METHOD FB_init : BOOL
VAR_INPUT
	bInitRetains : BOOL; // if TRUE, the retain variables are initialized (warm start / cold start)
	bInCopyCode : BOOL;  // if TRUE, the instance afterwards gets moved into the copy code (online change)
	InitialValue : ETcVnMorphologicalOperator;
END_VAR
localData := InitialValue;
AddBaseDatatype(enumBaseDatatype);
ClearReference();

AddLocalEnumeration('TCVN_MO_EROSION', ETcVnMorphologicalOperator.TCVN_MO_EROSION);
AddLocalEnumeration('TCVN_MO_DILATION', ETcVnMorphologicalOperator.TCVN_MO_DILATION);
AddLocalEnumeration('TCVN_MO_OPENING', ETcVnMorphologicalOperator.TCVN_MO_OPENING);
AddLocalEnumeration('TCVN_MO_CLOSING', ETcVnMorphologicalOperator.TCVN_MO_CLOSING);
AddLocalEnumeration('TCVN_MO_GRADIENT', ETcVnMorphologicalOperator.TCVN_MO_GRADIENT);
AddLocalEnumeration('TCVN_MO_WHITE_TOPHAT', .TCVN_MO_WHITE_TOPHAT);
AddLocalEnumeration('TCVN_MO_BLACK_TOPHAT', ETcVnMorphologicalOperator.TCVN_MO_BLACK_TOPHAT);
AddLocalEnumeration('TCVN_MO_OPENING_BY_RECONSTRUCTION', ETcVnMorphologicalOperator.TCVN_MO_OPENING_BY_RECONSTRUCTION);
AddLocalEnumeration('TCVN_MO_CLOSING_BY_RECONSTRUCTION', ETcVnMorphologicalOperator.TCVN_MO_CLOSING_BY_RECONSTRUCTION);
AddLocalEnumeration('TCVN_MO_WHITE_TOPHAT_BY_RECONSTRUCTION', ETcVnMorphologicalOperator.TCVN_MO_WHITE_TOPHAT_BY_RECONSTRUCTION);
AddLocalEnumeration('TCVN_MO_BLACK_TOPHAT_BY_RECONSTRUCTION', ETcVnMorphologicalOperator.TCVN_MO_BLACK_TOPHAT_BY_RECONSTRUCTION);
END_METHOD

PROPERTY PUBLIC Identifier : T_MAXSTRING
GET
Identifier := 'ETcVnMorphologicalOperator';
END_GET
END_PROPERTY

METHOD IsEnumeratorValueEqual : BOOL
VAR_INPUT
	Enumerator : I_KeyValueForwardEnumerator;
END_VAR
VAR
	storedValue : ETcVnMorphologicalOperator;
END_VAR
IF NOT Enumerator.TryGet(storedValue) THEN
	RETURN;
END_IF

IsEnumeratorValueEqual := storedValue = activeData;
END_METHOD

METHOD PUBLIC MakeReferenceTo
VAR_INPUT
	ReferenceTarget : REFERENCE TO ETcVnMorphologicalOperator;
END_VAR
activeData REF= ReferenceTarget;
SetBaseDatatypeReference();
END_METHOD

METHOD PROTECTED SetBaseDatatypeReference
VAR_INPUT
END_VAR
enumBaseDatatype.MakeReferenceTo(activeData);
END_METHOD

PROPERTY PUBLIC Size : UDINT
GET
Size := SIZEOF(activeData);
END_GET
END_PROPERTY

METHOD TryMakeReferenceTo : BOOL
VAR_INPUT
	Target : I_Datatype;
END_VAR
VAR
	targetAsEnum : I_EnumDatatype;
	pTargetData : POINTER TO ETcVnMorphologicalOperator;
END_VAR
IF NOT Target.TryResolveAsEnumDatatype(targetAsEnum) THEN
	RETURN;
END_IF

IF targetAsEnum.Identifier <> Identifier THEN
	RETURN;
END_IF

pTargetData := Target.Address;
activeData REF= pTargetData^;
SetBaseDatatypeReference();
TryMakeReferenceTo := TRUE;
END_METHOD

PROPERTY PUBLIC Value : ETcVnMorphologicalOperator
GET
Value := activeData;
END_GET
SET
activeData := Value;
END_SET
END_PROPERTY

END_FUNCTION_BLOCK

// ---- Enums/_ETcVnNbc.TcPOU
{attribute 'linkalways'} 
{attribute 'no_explicit_call' := 'This FB is a CLASS and must be accessed using methods or properties'}
{attribute 'enable_dynamic_creation'}
FUNCTION_BLOCK _ETcVnNbc EXTENDS EnumDatatypeBase
VAR
	localData : ETcVnNbc;
	activeData : REFERENCE TO ETcVnNbc;
	enumBaseDatatype : _UDINT(localData);
END_VAR

METHOD PRIVATE AddLocalEnumeration
VAR_INPUT
	Enumeration : T_MAXSTRING;
	Value : ETcVnNbc;
END_VAR
AddEnumeration(Enumeration, Value);
END_METHOD

PROPERTY PUBLIC Address : PVOID
GET
Address := ADR(activeData);
END_GET
END_PROPERTY

METHOD PUBLIC ClearReference
VAR_INPUT
END_VAR
activeData REF= localData;
SetBaseDatatypeReference();
END_METHOD

METHOD PUBLIC Clone : I_Datatype
VAR
    pClone : POINTER TO _ETcVnNbc;
END_VAR
pClone := __NEW(_ETcVnNbc(InitialValue := Value));
Clone := pClone^;
END_METHOD

METHOD FB_init : BOOL
VAR_INPUT
	bInitRetains : BOOL; // if TRUE, the retain variables are initialized (warm start / cold start)
	bInCopyCode : BOOL;  // if TRUE, the instance afterwards gets moved into the copy code (online change)
	InitialValue : ETcVnNbc;
END_VAR
localData := InitialValue;
AddBaseDatatype(enumBaseDatatype);
ClearReference();

AddLocalEnumeration('TCVN_NBC_CLASSIFIER', ETcVnNbc.TCVN_NBC_CLASSIFIER);
AddLocalEnumeration('TCVN_NBC_NOVELTY_DETECTOR', ETcVnNbc.TCVN_NBC_NOVELTY_DETECTOR);
END_METHOD

PROPERTY PUBLIC Identifier : T_MAXSTRING
GET
Identifier := 'ETcVnNbc';
END_GET
END_PROPERTY

METHOD IsEnumeratorValueEqual : BOOL
VAR_INPUT
	Enumerator : I_KeyValueForwardEnumerator;
END_VAR
VAR
	storedValue : ETcVnNbc;
END_VAR
IF NOT Enumerator.TryGet(storedValue) THEN
	RETURN;
END_IF

IsEnumeratorValueEqual := storedValue = activeData;
END_METHOD

METHOD PUBLIC MakeReferenceTo
VAR_INPUT
	ReferenceTarget : REFERENCE TO ETcVnNbc;
END_VAR
activeData REF= ReferenceTarget;
SetBaseDatatypeReference();
END_METHOD

METHOD PROTECTED SetBaseDatatypeReference
VAR_INPUT
END_VAR
enumBaseDatatype.MakeReferenceTo(activeData);
END_METHOD

PROPERTY PUBLIC Size : UDINT
GET
Size := SIZEOF(activeData);
END_GET
END_PROPERTY

METHOD TryMakeReferenceTo : BOOL
VAR_INPUT
	Target : I_Datatype;
END_VAR
VAR
	targetAsEnum : I_EnumDatatype;
	pTargetData : POINTER TO ETcVnNbc;
END_VAR
IF NOT Target.TryResolveAsEnumDatatype(targetAsEnum) THEN
	RETURN;
END_IF

IF targetAsEnum.Identifier <> Identifier THEN
	RETURN;
END_IF

pTargetData := Target.Address;
activeData REF= pTargetData^;
SetBaseDatatypeReference();
TryMakeReferenceTo := TRUE;
END_METHOD

PROPERTY PUBLIC Value : ETcVnNbc
GET
Value := activeData;
END_GET
SET
activeData := Value;
END_SET
END_PROPERTY

END_FUNCTION_BLOCK

// ---- Enums/_ETcVnNormalizationType.TcPOU
{attribute 'linkalways'} 
{attribute 'no_explicit_call' := 'This FB is a CLASS and must be accessed using methods or properties'}
{attribute 'enable_dynamic_creation'}
FUNCTION_BLOCK _ETcVnNormalizationType EXTENDS EnumDatatypeBase
VAR
	localData : ETcVnNormalizationType;
	activeData : REFERENCE TO ETcVnNormalizationType;
	enumBaseDatatype : _DINT(localData);
END_VAR

METHOD PRIVATE AddLocalEnumeration
VAR_INPUT
	Enumeration : T_MAXSTRING;
	Value : ETcVnNormalizationType;
END_VAR
AddEnumeration(Enumeration, Value);
END_METHOD

PROPERTY PUBLIC Address : PVOID
GET
Address := ADR(activeData);
END_GET
END_PROPERTY

METHOD PUBLIC ClearReference
VAR_INPUT
END_VAR
activeData REF= localData;
SetBaseDatatypeReference();
END_METHOD

METHOD PUBLIC Clone : I_Datatype
VAR
    pClone : POINTER TO _ETcVnNormalizationType;
END_VAR
pClone := __NEW(_ETcVnNormalizationType(InitialValue := Value));
Clone := pClone^;
END_METHOD

METHOD FB_init : BOOL
VAR_INPUT
	bInitRetains : BOOL; // if TRUE, the retain variables are initialized (warm start / cold start)
	bInCopyCode : BOOL;  // if TRUE, the instance afterwards gets moved into the copy code (online change)
	InitialValue : ETcVnNormalizationType;
END_VAR
localData := InitialValue;
AddBaseDatatype(enumBaseDatatype);
ClearReference();

AddLocalEnumeration('TCVN_NT_INF', ETcVnNormalizationType.TCVN_NT_INF);
AddLocalEnumeration('TCVN_NT_L1', ETcVnNormalizationType.TCVN_NT_L1);
AddLocalEnumeration('TCVN_NT_L2', ETcVnNormalizationType.TCVN_NT_L2);
AddLocalEnumeration('TCVN_NT_L2SQR', ETcVnNormalizationType.TCVN_NT_L2SQR);
AddLocalEnumeration('TCVN_NT_HAMMING', ETcVnNormalizationType.TCVN_NT_HAMMING);
AddLocalEnumeration('TCVN_NT_HAMMING2', ETcVnNormalizationType.TCVN_NT_HAMMING2);
AddLocalEnumeration('TCVN_NT_RELATIVE_INF', ETcVnNormalizationType.TCVN_NT_RELATIVE_INF);
AddLocalEnumeration('TCVN_NT_RELATIVE_L1', ETcVnNormalizationType.TCVN_NT_RELATIVE_L1);
AddLocalEnumeration('TCVN_NT_RELATIVE_L2', ETcVnNormalizationType.TCVN_NT_RELATIVE_L2);
AddLocalEnumeration('TCVN_NT_RELATIVE_L2SQR', ETcVnNormalizationType.TCVN_NT_RELATIVE_L2SQR);
AddLocalEnumeration('TCVN_NT_RELATIVE_HAMMING', ETcVnNormalizationType.TCVN_NT_RELATIVE_HAMMING);
AddLocalEnumeration('TCVN_NT_RELATIVE_HAMMING2', ETcVnNormalizationType.TCVN_NT_RELATIVE_HAMMING2);
AddLocalEnumeration('TCVN_NT_MINMAX', ETcVnNormalizationType.TCVN_NT_MINMAX);
END_METHOD

PROPERTY PUBLIC Identifier : T_MAXSTRING
GET
Identifier := 'ETcVnNormalizationType';
END_GET
END_PROPERTY

METHOD IsEnumeratorValueEqual : BOOL
VAR_INPUT
	Enumerator : I_KeyValueForwardEnumerator;
END_VAR
VAR
	storedValue : ETcVnNormalizationType;
END_VAR
IF NOT Enumerator.TryGet(storedValue) THEN
	RETURN;
END_IF

IsEnumeratorValueEqual := storedValue = activeData;
END_METHOD

METHOD PUBLIC MakeReferenceTo
VAR_INPUT
	ReferenceTarget : REFERENCE TO ETcVnNormalizationType;
END_VAR
activeData REF= ReferenceTarget;
SetBaseDatatypeReference();
END_METHOD

METHOD PROTECTED SetBaseDatatypeReference
VAR_INPUT
END_VAR
enumBaseDatatype.MakeReferenceTo(activeData);
END_METHOD

PROPERTY PUBLIC Size : UDINT
GET
Size := SIZEOF(activeData);
END_GET
END_PROPERTY

METHOD TryMakeReferenceTo : BOOL
VAR_INPUT
	Target : I_Datatype;
END_VAR
VAR
	targetAsEnum : I_EnumDatatype;
	pTargetData : POINTER TO ETcVnNormalizationType;
END_VAR
IF NOT Target.TryResolveAsEnumDatatype(targetAsEnum) THEN
	RETURN;
END_IF

IF targetAsEnum.Identifier <> Identifier THEN
	RETURN;
END_IF

pTargetData := Target.Address;
activeData REF= pTargetData^;
SetBaseDatatypeReference();
TryMakeReferenceTo := TRUE;
END_METHOD

PROPERTY PUBLIC Value : ETcVnNormalizationType
GET
Value := activeData;
END_GET
SET
activeData := Value;
END_SET
END_PROPERTY

END_FUNCTION_BLOCK

// ---- Enums/_ETcVnOcrModelType.TcPOU
{attribute 'linkalways'} 
{attribute 'no_explicit_call' := 'This FB is a CLASS and must be accessed using methods or properties'}
{attribute 'enable_dynamic_creation'}
FUNCTION_BLOCK _ETcVnOcrModelType EXTENDS EnumDatatypeBase
VAR
	localData : ETcVnOcrModelType;
	activeData : REFERENCE TO ETcVnOcrModelType;
	enumBaseDatatype : _ULINT(localData);
END_VAR

METHOD PRIVATE AddLocalEnumeration
VAR_INPUT
	Enumeration : T_MAXSTRING;
	Value : ETcVnOcrModelType;
END_VAR
AddEnumeration(Enumeration, Value);
END_METHOD

PROPERTY PUBLIC Address : PVOID
GET
Address := ADR(activeData);
END_GET
END_PROPERTY

METHOD PUBLIC ClearReference
VAR_INPUT
END_VAR
activeData REF= localData;
SetBaseDatatypeReference();
END_METHOD

METHOD PUBLIC Clone : I_Datatype
VAR
    pClone : POINTER TO _ETcVnOcrModelType;
END_VAR
pClone := __NEW(_ETcVnOcrModelType(InitialValue := Value));
Clone := pClone^;
END_METHOD

METHOD FB_init : BOOL
VAR_INPUT
	bInitRetains : BOOL; // if TRUE, the retain variables are initialized (warm start / cold start)
	bInCopyCode : BOOL;  // if TRUE, the instance afterwards gets moved into the copy code (online change)
	InitialValue : ETcVnOcrModelType;
END_VAR
localData := InitialValue;
AddBaseDatatype(enumBaseDatatype);
ClearReference();

AddLocalEnumeration('TCVN_OMT_NUMBERS', ETcVnOcrModelType.TCVN_OMT_NUMBERS);
AddLocalEnumeration('TCVN_OMT_NUMBERS_SC', ETcVnOcrModelType.TCVN_OMT_NUMBERS_SC);
AddLocalEnumeration('TCVN_OMT_UCLETTERS', ETcVnOcrModelType.TCVN_OMT_UCLETTERS);
AddLocalEnumeration('TCVN_OMT_NUMBERS_SC_UCLETTERS', ETcVnOcrModelType.TCVN_OMT_NUMBERS_SC_UCLETTERS);
END_METHOD

PROPERTY PUBLIC Identifier : T_MAXSTRING
GET
Identifier := 'ETcVnOcrModelType';
END_GET
END_PROPERTY

METHOD IsEnumeratorValueEqual : BOOL
VAR_INPUT
	Enumerator : I_KeyValueForwardEnumerator;
END_VAR
VAR
	storedValue : ETcVnOcrModelType;
END_VAR
IF NOT Enumerator.TryGet(storedValue) THEN
	RETURN;
END_IF

IsEnumeratorValueEqual := storedValue = activeData;
END_METHOD

METHOD PUBLIC MakeReferenceTo
VAR_INPUT
	ReferenceTarget : REFERENCE TO ETcVnOcrModelType;
END_VAR
activeData REF= ReferenceTarget;
SetBaseDatatypeReference();
END_METHOD

METHOD PROTECTED SetBaseDatatypeReference
VAR_INPUT
END_VAR
enumBaseDatatype.MakeReferenceTo(activeData);
END_METHOD

PROPERTY PUBLIC Size : UDINT
GET
Size := SIZEOF(activeData);
END_GET
END_PROPERTY

METHOD TryMakeReferenceTo : BOOL
VAR_INPUT
	Target : I_Datatype;
END_VAR
VAR
	targetAsEnum : I_EnumDatatype;
	pTargetData : POINTER TO ETcVnOcrModelType;
END_VAR
IF NOT Target.TryResolveAsEnumDatatype(targetAsEnum) THEN
	RETURN;
END_IF

IF targetAsEnum.Identifier <> Identifier THEN
	RETURN;
END_IF

pTargetData := Target.Address;
activeData REF= pTargetData^;
SetBaseDatatypeReference();
TryMakeReferenceTo := TRUE;
END_METHOD

PROPERTY PUBLIC Value : ETcVnOcrModelType
GET
Value := activeData;
END_GET
SET
activeData := Value;
END_SET
END_PROPERTY

END_FUNCTION_BLOCK

// ---- Enums/_ETcVnOcrOptions.TcPOU
{attribute 'linkalways'} 
{attribute 'no_explicit_call' := 'This FB is a CLASS and must be accessed using methods or properties'}
{attribute 'enable_dynamic_creation'}
FUNCTION_BLOCK _ETcVnOcrOptions EXTENDS EnumDatatypeBase
VAR
	localData : ETcVnOcrOptions;
	activeData : REFERENCE TO ETcVnOcrOptions;
	enumBaseDatatype : _UDINT(localData);
END_VAR

METHOD PRIVATE AddLocalEnumeration
VAR_INPUT
	Enumeration : T_MAXSTRING;
	Value : ETcVnOcrOptions;
END_VAR
AddEnumeration(Enumeration, Value);
END_METHOD

PROPERTY PUBLIC Address : PVOID
GET
Address := ADR(activeData);
END_GET
END_PROPERTY

METHOD PUBLIC ClearReference
VAR_INPUT
END_VAR
activeData REF= localData;
SetBaseDatatypeReference();
END_METHOD

METHOD PUBLIC Clone : I_Datatype
VAR
    pClone : POINTER TO _ETcVnOcrOptions;
END_VAR
pClone := __NEW(_ETcVnOcrOptions(InitialValue := Value));
Clone := pClone^;
END_METHOD

METHOD FB_init : BOOL
VAR_INPUT
	bInitRetains : BOOL; // if TRUE, the retain variables are initialized (warm start / cold start)
	bInCopyCode : BOOL;  // if TRUE, the instance afterwards gets moved into the copy code (online change)
	InitialValue : ETcVnOcrOptions;
END_VAR
localData := InitialValue;
AddBaseDatatype(enumBaseDatatype);
ClearReference();

AddLocalEnumeration('TCVN_OO_WITHBLANKS', ETcVnOcrOptions.TCVN_OO_WITHBLANKS);
END_METHOD

PROPERTY PUBLIC Identifier : T_MAXSTRING
GET
Identifier := 'ETcVnOcrOptions';
END_GET
END_PROPERTY

METHOD IsEnumeratorValueEqual : BOOL
VAR_INPUT
	Enumerator : I_KeyValueForwardEnumerator;
END_VAR
VAR
	storedValue : ETcVnOcrOptions;
END_VAR
IF NOT Enumerator.TryGet(storedValue) THEN
	RETURN;
END_IF

IsEnumeratorValueEqual := storedValue = activeData;
END_METHOD

METHOD PUBLIC MakeReferenceTo
VAR_INPUT
	ReferenceTarget : REFERENCE TO ETcVnOcrOptions;
END_VAR
activeData REF= ReferenceTarget;
SetBaseDatatypeReference();
END_METHOD

METHOD PROTECTED SetBaseDatatypeReference
VAR_INPUT
END_VAR
enumBaseDatatype.MakeReferenceTo(activeData);
END_METHOD

PROPERTY PUBLIC Size : UDINT
GET
Size := SIZEOF(activeData);
END_GET
END_PROPERTY

METHOD TryMakeReferenceTo : BOOL
VAR_INPUT
	Target : I_Datatype;
END_VAR
VAR
	targetAsEnum : I_EnumDatatype;
	pTargetData : POINTER TO ETcVnOcrOptions;
END_VAR
IF NOT Target.TryResolveAsEnumDatatype(targetAsEnum) THEN
	RETURN;
END_IF

IF targetAsEnum.Identifier <> Identifier THEN
	RETURN;
END_IF

pTargetData := Target.Address;
activeData REF= pTargetData^;
SetBaseDatatypeReference();
TryMakeReferenceTo := TRUE;
END_METHOD

PROPERTY PUBLIC Value : ETcVnOcrOptions
GET
Value := activeData;
END_GET
SET
activeData := Value;
END_SET
END_PROPERTY

END_FUNCTION_BLOCK

// ---- Enums/_ETcVnOrientationMethod.TcPOU
{attribute 'linkalways'} 
{attribute 'no_explicit_call' := 'This FB is a CLASS and must be accessed using methods or properties'}
{attribute 'enable_dynamic_creation'}
FUNCTION_BLOCK _ETcVnOrientationMethod EXTENDS EnumDatatypeBase
VAR
	localData : ETcVnOrientationMethod;
	activeData : REFERENCE TO ETcVnOrientationMethod;
	enumBaseDatatype : _DINT(localData);
END_VAR

METHOD PRIVATE AddLocalEnumeration
VAR_INPUT
	Enumeration : T_MAXSTRING;
	Value : ETcVnOrientationMethod;
END_VAR
AddEnumeration(Enumeration, Value);
END_METHOD

PROPERTY PUBLIC Address : PVOID
GET
Address := ADR(activeData);
END_GET
END_PROPERTY

METHOD PUBLIC ClearReference
VAR_INPUT
END_VAR
activeData REF= localData;
SetBaseDatatypeReference();
END_METHOD

METHOD PUBLIC Clone : I_Datatype
VAR
    pClone : POINTER TO _ETcVnOrientationMethod;
END_VAR
pClone := __NEW(_ETcVnOrientationMethod(InitialValue := Value));
Clone := pClone^;
END_METHOD

METHOD FB_init : BOOL
VAR_INPUT
	bInitRetains : BOOL; // if TRUE, the retain variables are initialized (warm start / cold start)
	bInCopyCode : BOOL;  // if TRUE, the instance afterwards gets moved into the copy code (online change)
	InitialValue : ETcVnOrientationMethod;
END_VAR
localData := InitialValue;
AddBaseDatatype(enumBaseDatatype);
ClearReference();

AddLocalEnumeration('TCVN_OM_PCA', ETcVnOrientationMethod.TCVN_OM_PCA);
AddLocalEnumeration('TCVN_OM_FITELLIPSE', ETcVnOrientationMethod.TCVN_OM_FITELLIPSE);
AddLocalEnumeration('TCVN_OM_MOMENTS', ETcVnOrientationMethod.TCVN_OM_MOMENTS);
AddLocalEnumeration('TCVN_OM_ENCLOSINGRECT', ETcVnOrientationMethod.TCVN_OM_ENCLOSINGRECT);
END_METHOD

PROPERTY PUBLIC Identifier : T_MAXSTRING
GET
Identifier := 'ETcVnOrientationMethod';
END_GET
END_PROPERTY

METHOD IsEnumeratorValueEqual : BOOL
VAR_INPUT
	Enumerator : I_KeyValueForwardEnumerator;
END_VAR
VAR
	storedValue : ETcVnOrientationMethod;
END_VAR
IF NOT Enumerator.TryGet(storedValue) THEN
	RETURN;
END_IF

IsEnumeratorValueEqual := storedValue = activeData;
END_METHOD

METHOD PUBLIC MakeReferenceTo
VAR_INPUT
	ReferenceTarget : REFERENCE TO ETcVnOrientationMethod;
END_VAR
activeData REF= ReferenceTarget;
SetBaseDatatypeReference();
END_METHOD

METHOD PROTECTED SetBaseDatatypeReference
VAR_INPUT
END_VAR
enumBaseDatatype.MakeReferenceTo(activeData);
END_METHOD

PROPERTY PUBLIC Size : UDINT
GET
Size := SIZEOF(activeData);
END_GET
END_PROPERTY

METHOD TryMakeReferenceTo : BOOL
VAR_INPUT
	Target : I_Datatype;
END_VAR
VAR
	targetAsEnum : I_EnumDatatype;
	pTargetData : POINTER TO ETcVnOrientationMethod;
END_VAR
IF NOT Target.TryResolveAsEnumDatatype(targetAsEnum) THEN
	RETURN;
END_IF

IF targetAsEnum.Identifier <> Identifier THEN
	RETURN;
END_IF

pTargetData := Target.Address;
activeData REF= pTargetData^;
SetBaseDatatypeReference();
TryMakeReferenceTo := TRUE;
END_METHOD

PROPERTY PUBLIC Value : ETcVnOrientationMethod
GET
Value := activeData;
END_GET
SET
activeData := Value;
END_SET
END_PROPERTY

END_FUNCTION_BLOCK

// ---- Enums/_ETcVnPaddingMode.TcPOU
{attribute 'linkalways'} 
{attribute 'no_explicit_call' := 'This FB is a CLASS and must be accessed using methods or properties'}
{attribute 'enable_dynamic_creation'}
FUNCTION_BLOCK _ETcVnPaddingMode EXTENDS EnumDatatypeBase
VAR
	localData : ETcVnPaddingMode;
	activeData : REFERENCE TO ETcVnPaddingMode;
	enumBaseDatatype : _DINT(localData);
END_VAR

METHOD PRIVATE AddLocalEnumeration
VAR_INPUT
	Enumeration : T_MAXSTRING;
	Value : ETcVnPaddingMode;
END_VAR
AddEnumeration(Enumeration, Value);
END_METHOD

PROPERTY PUBLIC Address : PVOID
GET
Address := ADR(activeData);
END_GET
END_PROPERTY

METHOD PUBLIC ClearReference
VAR_INPUT
END_VAR
activeData REF= localData;
SetBaseDatatypeReference();
END_METHOD

METHOD PUBLIC Clone : I_Datatype
VAR
    pClone : POINTER TO _ETcVnPaddingMode;
END_VAR
pClone := __NEW(_ETcVnPaddingMode(InitialValue := Value));
Clone := pClone^;
END_METHOD

METHOD FB_init : BOOL
VAR_INPUT
	bInitRetains : BOOL; // if TRUE, the retain variables are initialized (warm start / cold start)
	bInCopyCode : BOOL;  // if TRUE, the instance afterwards gets moved into the copy code (online change)
	InitialValue : ETcVnPaddingMode;
END_VAR
localData := InitialValue;
AddBaseDatatype(enumBaseDatatype);
ClearReference();

AddLocalEnumeration('TCVN_PM_NONE', ETcVnPaddingMode.TCVN_PM_NONE);
AddLocalEnumeration('TCVN_PM_CROP_CENTER', ETcVnPaddingMode.TCVN_PM_CROP_CENTER);
AddLocalEnumeration('TCVN_PM_LETTERBOX', ETcVnPaddingMode.TCVN_PM_LETTERBOX);
END_METHOD

PROPERTY PUBLIC Identifier : T_MAXSTRING
GET
Identifier := 'ETcVnPaddingMode';
END_GET
END_PROPERTY

METHOD IsEnumeratorValueEqual : BOOL
VAR_INPUT
	Enumerator : I_KeyValueForwardEnumerator;
END_VAR
VAR
	storedValue : ETcVnPaddingMode;
END_VAR
IF NOT Enumerator.TryGet(storedValue) THEN
	RETURN;
END_IF

IsEnumeratorValueEqual := storedValue = activeData;
END_METHOD

METHOD PUBLIC MakeReferenceTo
VAR_INPUT
	ReferenceTarget : REFERENCE TO ETcVnPaddingMode;
END_VAR
activeData REF= ReferenceTarget;
SetBaseDatatypeReference();
END_METHOD

METHOD PROTECTED SetBaseDatatypeReference
VAR_INPUT
END_VAR
enumBaseDatatype.MakeReferenceTo(activeData);
END_METHOD

PROPERTY PUBLIC Size : UDINT
GET
Size := SIZEOF(activeData);
END_GET
END_PROPERTY

METHOD TryMakeReferenceTo : BOOL
VAR_INPUT
	Target : I_Datatype;
END_VAR
VAR
	targetAsEnum : I_EnumDatatype;
	pTargetData : POINTER TO ETcVnPaddingMode;
END_VAR
IF NOT Target.TryResolveAsEnumDatatype(targetAsEnum) THEN
	RETURN;
END_IF

IF targetAsEnum.Identifier <> Identifier THEN
	RETURN;
END_IF

pTargetData := Target.Address;
activeData REF= pTargetData^;
SetBaseDatatypeReference();
TryMakeReferenceTo := TRUE;
END_METHOD

PROPERTY PUBLIC Value : ETcVnPaddingMode
GET
Value := activeData;
END_GET
SET
activeData := Value;
END_SET
END_PROPERTY

END_FUNCTION_BLOCK

// ---- Enums/_ETcVnPixelConnectivity.TcPOU
{attribute 'linkalways'} 
{attribute 'no_explicit_call' := 'This FB is a CLASS and must be accessed using methods or properties'}
{attribute 'enable_dynamic_creation'}
FUNCTION_BLOCK _ETcVnPixelConnectivity EXTENDS EnumDatatypeBase
VAR
	localData : ETcVnPixelConnectivity;
	activeData : REFERENCE TO ETcVnPixelConnectivity;
	enumBaseDatatype : _DINT(localData);
END_VAR

METHOD PRIVATE AddLocalEnumeration
VAR_INPUT
	Enumeration : T_MAXSTRING;
	Value : ETcVnPixelConnectivity;
END_VAR
AddEnumeration(Enumeration, Value);
END_METHOD

PROPERTY PUBLIC Address : PVOID
GET
Address := ADR(activeData);
END_GET
END_PROPERTY

METHOD PUBLIC ClearReference
VAR_INPUT
END_VAR
activeData REF= localData;
SetBaseDatatypeReference();
END_METHOD

METHOD PUBLIC Clone : I_Datatype
VAR
    pClone : POINTER TO _ETcVnPixelConnectivity;
END_VAR
pClone := __NEW(_ETcVnPixelConnectivity(InitialValue := Value));
Clone := pClone^;
END_METHOD

METHOD FB_init : BOOL
VAR_INPUT
	bInitRetains : BOOL; // if TRUE, the retain variables are initialized (warm start / cold start)
	bInCopyCode : BOOL;  // if TRUE, the instance afterwards gets moved into the copy code (online change)
	InitialValue : ETcVnPixelConnectivity;
END_VAR
localData := InitialValue;
AddBaseDatatype(enumBaseDatatype);
ClearReference();

AddLocalEnumeration('TCVN_PC_4', ETcVnPixelConnectivity.TCVN_PC_4);
AddLocalEnumeration('TCVN_PC_8', ETcVnPixelConnectivity.TCVN_PC_8);
END_METHOD

PROPERTY PUBLIC Identifier : T_MAXSTRING
GET
Identifier := 'ETcVnPixelConnectivity';
END_GET
END_PROPERTY

METHOD IsEnumeratorValueEqual : BOOL
VAR_INPUT
	Enumerator : I_KeyValueForwardEnumerator;
END_VAR
VAR
	storedValue : ETcVnPixelConnectivity;
END_VAR
IF NOT Enumerator.TryGet(storedValue) THEN
	RETURN;
END_IF

IsEnumeratorValueEqual := storedValue = activeData;
END_METHOD

METHOD PUBLIC MakeReferenceTo
VAR_INPUT
	ReferenceTarget : REFERENCE TO ETcVnPixelConnectivity;
END_VAR
activeData REF= ReferenceTarget;
SetBaseDatatypeReference();
END_METHOD

METHOD PROTECTED SetBaseDatatypeReference
VAR_INPUT
END_VAR
enumBaseDatatype.MakeReferenceTo(activeData);
END_METHOD

PROPERTY PUBLIC Size : UDINT
GET
Size := SIZEOF(activeData);
END_GET
END_PROPERTY

METHOD TryMakeReferenceTo : BOOL
VAR_INPUT
	Target : I_Datatype;
END_VAR
VAR
	targetAsEnum : I_EnumDatatype;
	pTargetData : POINTER TO ETcVnPixelConnectivity;
END_VAR
IF NOT Target.TryResolveAsEnumDatatype(targetAsEnum) THEN
	RETURN;
END_IF

IF targetAsEnum.Identifier <> Identifier THEN
	RETURN;
END_IF

pTargetData := Target.Address;
activeData REF= pTargetData^;
SetBaseDatatypeReference();
TryMakeReferenceTo := TRUE;
END_METHOD

PROPERTY PUBLIC Value : ETcVnPixelConnectivity
GET
Value := activeData;
END_GET
SET
activeData := Value;
END_SET
END_PROPERTY

END_FUNCTION_BLOCK

// ---- Enums/_ETcVnPixelEncoding.TcPOU
{attribute 'linkalways'} 
{attribute 'no_explicit_call' := 'This FB is a CLASS and must be accessed using methods or properties'}
{attribute 'enable_dynamic_creation'}
FUNCTION_BLOCK _ETcVnPixelEncoding EXTENDS EnumDatatypeBase
VAR
	localData : ETcVnPixelEncoding;
	activeData : REFERENCE TO ETcVnPixelEncoding;
	enumBaseDatatype : _BYTE(localData);
END_VAR

METHOD PRIVATE AddLocalEnumeration
VAR_INPUT
	Enumeration : T_MAXSTRING;
	Value : ETcVnPixelEncoding;
END_VAR
AddEnumeration(Enumeration, Value);
END_METHOD

PROPERTY PUBLIC Address : PVOID
GET
Address := ADR(activeData);
END_GET
END_PROPERTY

METHOD PUBLIC ClearReference
VAR_INPUT
END_VAR
activeData REF= localData;
SetBaseDatatypeReference();
END_METHOD

METHOD PUBLIC Clone : I_Datatype
VAR
    pClone : POINTER TO _ETcVnPixelEncoding;
END_VAR
pClone := __NEW(_ETcVnPixelEncoding(InitialValue := Value));
Clone := pClone^;
END_METHOD

METHOD FB_init : BOOL
VAR_INPUT
	bInitRetains : BOOL; // if TRUE, the retain variables are initialized (warm start / cold start)
	bInCopyCode : BOOL;  // if TRUE, the instance afterwards gets moved into the copy code (online change)
	InitialValue : ETcVnPixelEncoding;
END_VAR
localData := InitialValue;
AddBaseDatatype(enumBaseDatatype);
ClearReference();

AddLocalEnumeration('TCVN_PE_NONE', ETcVnPixelEncoding.TCVN_PE_NONE);
AddLocalEnumeration('TCVN_PE_BAYER_GR', ETcVnPixelEncoding.TCVN_PE_BAYER_GR);
AddLocalEnumeration('TCVN_PE_BAYER_RG', ETcVnPixelEncoding.TCVN_PE_BAYER_RG);
AddLocalEnumeration('TCVN_PE_BAYER_GB', ETcVnPixelEncoding.TCVN_PE_BAYER_GB);
AddLocalEnumeration('TCVN_PE_BAYER_BG', ETcVnPixelEncoding.TCVN_PE_BAYER_BG);
AddLocalEnumeration('TCVN_PE_YUV_411_UYYVYY', ETcVnPixelEncoding.TCVN_PE_YUV_411_UYYVYY);
AddLocalEnumeration('TCVN_PE_YUV_422_UYVY', ETcVnPixelEncoding.TCVN_PE_YUV_422_UYVY);
AddLocalEnumeration('TCVN_PE_YUV_422_YUYV', ETcVnPixelEncoding.TCVN_PE_YUV_422_YUYV);
AddLocalEnumeration('TCVN_PE_YCBCR_411_CBYYCRYY', ETcVnPixelEncoding.TCVN_PE_YCBCR_411_CBYYCRYY);
AddLocalEnumeration('TCVN_PE_YCBCR_422_CBYCRY', ETcVnPixelEncoding.TCVN_PE_YCBCR_422_CBYCRY);
AddLocalEnumeration('TCVN_PE_YCBCR_422_YCBYCR', ETcVnPixelEncoding.TCVN_PE_YCBCR_422_YCBYCR);
END_METHOD

PROPERTY PUBLIC Identifier : T_MAXSTRING
GET
Identifier := 'ETcVnPixelEncoding';
END_GET
END_PROPERTY

METHOD IsEnumeratorValueEqual : BOOL
VAR_INPUT
	Enumerator : I_KeyValueForwardEnumerator;
END_VAR
VAR
	storedValue : ETcVnPixelEncoding;
END_VAR
IF NOT Enumerator.TryGet(storedValue) THEN
	RETURN;
END_IF

IsEnumeratorValueEqual := storedValue = activeData;
END_METHOD

METHOD PUBLIC MakeReferenceTo
VAR_INPUT
	ReferenceTarget : REFERENCE TO ETcVnPixelEncoding;
END_VAR
activeData REF= ReferenceTarget;
SetBaseDatatypeReference();
END_METHOD

METHOD PROTECTED SetBaseDatatypeReference
VAR_INPUT
END_VAR
enumBaseDatatype.MakeReferenceTo(activeData);
END_METHOD

PROPERTY PUBLIC Size : UDINT
GET
Size := SIZEOF(activeData);
END_GET
END_PROPERTY

METHOD TryMakeReferenceTo : BOOL
VAR_INPUT
	Target : I_Datatype;
END_VAR
VAR
	targetAsEnum : I_EnumDatatype;
	pTargetData : POINTER TO ETcVnPixelEncoding;
END_VAR
IF NOT Target.TryResolveAsEnumDatatype(targetAsEnum) THEN
	RETURN;
END_IF

IF targetAsEnum.Identifier <> Identifier THEN
	RETURN;
END_IF

pTargetData := Target.Address;
activeData REF= pTargetData^;
SetBaseDatatypeReference();
TryMakeReferenceTo := TRUE;
END_METHOD

PROPERTY PUBLIC Value : ETcVnPixelEncoding
GET
Value := activeData;
END_GET
SET
activeData := Value;
END_SET
END_PROPERTY

END_FUNCTION_BLOCK

// ---- Enums/_ETcVnColorMapSize.TcPOU
{attribute 'linkalways'} 
{attribute 'no_explicit_call' := 'This FB is a CLASS and must be accessed using methods or properties'}
{attribute 'enable_dynamic_creation'}
FUNCTION_BLOCK _ETcVnColorMapSize EXTENDS EnumDatatypeBase
VAR
	localData : ETcVnColorMapSize;
	activeData : REFERENCE TO ETcVnColorMapSize;
	enumBaseDatatype : _UDINT(localData);
END_VAR

METHOD PRIVATE AddLocalEnumeration
VAR_INPUT
	Enumeration : T_MAXSTRING;
	Value : ETcVnColorMapSize;
END_VAR
AddEnumeration(Enumeration, Value);
END_METHOD

PROPERTY PUBLIC Address : PVOID
GET
Address := ADR(activeData);
END_GET
END_PROPERTY

METHOD PUBLIC ClearReference
VAR_INPUT
END_VAR
activeData REF= localData;
SetBaseDatatypeReference();
END_METHOD

METHOD PUBLIC Clone : I_Datatype
VAR
    pClone : POINTER TO _ETcVnColorMapSize;
END_VAR
pClone := __NEW(_ETcVnColorMapSize(InitialValue := Value));
Clone := pClone^;
END_METHOD

METHOD FB_init : BOOL
VAR_INPUT
	bInitRetains : BOOL; // if TRUE, the retain variables are initialized (warm start / cold start)
	bInCopyCode : BOOL;  // if TRUE, the instance afterwards gets moved into the copy code (online change)
	InitialValue : ETcVnColorMapSize;
END_VAR
localData := InitialValue;
AddBaseDatatype(enumBaseDatatype);
ClearReference();

AddLocalEnumeration('TCVN_CMS_256', ETcVnColorMapSize.TCVN_CMS_256);
AddLocalEnumeration('TCVN_CMS_65536', ETcVnColorMapSize.TCVN_CMS_65536);
END_METHOD

PROPERTY PUBLIC Identifier : T_MAXSTRING
GET
Identifier := 'ETcVnColorMapSize';
END_GET
END_PROPERTY

METHOD IsEnumeratorValueEqual : BOOL
VAR_INPUT
	Enumerator : I_KeyValueForwardEnumerator;
END_VAR
VAR
	storedValue : ETcVnColorMapSize;
END_VAR
IF NOT Enumerator.TryGet(storedValue) THEN
	RETURN;
END_IF

IsEnumeratorValueEqual := storedValue = activeData;
END_METHOD

METHOD PUBLIC MakeReferenceTo
VAR_INPUT
	ReferenceTarget : REFERENCE TO ETcVnColorMapSize;
END_VAR
activeData REF= ReferenceTarget;
SetBaseDatatypeReference();
END_METHOD

METHOD PROTECTED SetBaseDatatypeReference
VAR_INPUT
END_VAR
enumBaseDatatype.MakeReferenceTo(activeData);
END_METHOD

PROPERTY PUBLIC Size : UDINT
GET
Size := SIZEOF(activeData);
END_GET
END_PROPERTY

METHOD TryMakeReferenceTo : BOOL
VAR_INPUT
	Target : I_Datatype;
END_VAR
VAR
	targetAsEnum : I_EnumDatatype;
	pTargetData : POINTER TO ETcVnColorMapSize;
END_VAR
IF NOT Target.TryResolveAsEnumDatatype(targetAsEnum) THEN
	RETURN;
END_IF

IF targetAsEnum.Identifier <> Identifier THEN
	RETURN;
END_IF

pTargetData := Target.Address;
activeData REF= pTargetData^;
SetBaseDatatypeReference();
TryMakeReferenceTo := TRUE;
END_METHOD

PROPERTY PUBLIC Value : ETcVnColorMapSize
GET
Value := activeData;
END_GET
SET
activeData := Value;
END_SET
END_PROPERTY

END_FUNCTION_BLOCK

// ---- Enums/_ETcVnAdaptiveThresholdMethod.TcPOU
{attribute 'linkalways'} 
{attribute 'no_explicit_call' := 'This FB is a CLASS and must be accessed using methods or properties'}
{attribute 'enable_dynamic_creation'}
FUNCTION_BLOCK _ETcVnAdaptiveThresholdMethod EXTENDS EnumDatatypeBase
VAR
	localData : ETcVnAdaptiveThresholdMethod;
	activeData : REFERENCE TO ETcVnAdaptiveThresholdMethod;
	enumBaseDatatype : _DINT(localData);
END_VAR

METHOD PRIVATE AddLocalEnumeration
VAR_INPUT
	Enumeration : T_MAXSTRING;
	Value : ETcVnAdaptiveThresholdMethod;
END_VAR
AddEnumeration(Enumeration, Value);
END_METHOD

PROPERTY PUBLIC Address : PVOID
GET
Address := ADR(activeData);
END_GET
END_PROPERTY

METHOD PUBLIC ClearReference
VAR_INPUT
END_VAR
activeData REF= localData;
SetBaseDatatypeReference();
END_METHOD

METHOD PUBLIC Clone : I_Datatype
VAR
    pClone : POINTER TO _ETcVnAdaptiveThresholdMethod;
END_VAR
pClone := __NEW(_ETcVnAdaptiveThresholdMethod(InitialValue := Value));
Clone := pClone^;
END_METHOD

METHOD FB_init : BOOL
VAR_INPUT
	bInitRetains : BOOL; // if TRUE, the retain variables are initialized (warm start / cold start)
	bInCopyCode : BOOL;  // if TRUE, the instance afterwards gets moved into the copy code (online change)
	InitialValue : ETcVnAdaptiveThresholdMethod;
END_VAR
localData := InitialValue;
AddBaseDatatype(enumBaseDatatype);
ClearReference();

AddLocalEnumeration('TCVN_ATM_MEAN', ETcVnAdaptiveThresholdMethod.TCVN_ATM_MEAN);
AddLocalEnumeration('TCVN_ATM_GAUSSIAN', ETcVnAdaptiveThresholdMethod.TCVN_ATM_GAUSSIAN);
END_METHOD

PROPERTY PUBLIC Identifier : T_MAXSTRING
GET
Identifier := 'ETcVnAdaptiveThresholdMethod';
END_GET
END_PROPERTY

METHOD IsEnumeratorValueEqual : BOOL
VAR_INPUT
	Enumerator : I_KeyValueForwardEnumerator;
END_VAR
VAR
	storedValue : ETcVnAdaptiveThresholdMethod;
END_VAR
IF NOT Enumerator.TryGet(storedValue) THEN
	RETURN;
END_IF

IsEnumeratorValueEqual := storedValue = activeData;
END_METHOD

METHOD PUBLIC MakeReferenceTo
VAR_INPUT
	ReferenceTarget : REFERENCE TO ETcVnAdaptiveThresholdMethod;
END_VAR
activeData REF= ReferenceTarget;
SetBaseDatatypeReference();
END_METHOD

METHOD PROTECTED SetBaseDatatypeReference
VAR_INPUT
END_VAR
enumBaseDatatype.MakeReferenceTo(activeData);
END_METHOD

PROPERTY PUBLIC Size : UDINT
GET
Size := SIZEOF(activeData);
END_GET
END_PROPERTY

METHOD TryMakeReferenceTo : BOOL
VAR_INPUT
	Target : I_Datatype;
END_VAR
VAR
	targetAsEnum : I_EnumDatatype;
	pTargetData : POINTER TO ETcVnAdaptiveThresholdMethod;
END_VAR
IF NOT Target.TryResolveAsEnumDatatype(targetAsEnum) THEN
	RETURN;
END_IF

IF targetAsEnum.Identifier <> Identifier THEN
	RETURN;
END_IF

pTargetData := Target.Address;
activeData REF= pTargetData^;
SetBaseDatatypeReference();
TryMakeReferenceTo := TRUE;
END_METHOD

PROPERTY PUBLIC Value : ETcVnAdaptiveThresholdMethod
GET
Value := activeData;
END_GET
SET
activeData := Value;
END_SET
END_PROPERTY

END_FUNCTION_BLOCK

// ---- Enums/_ETcVnCalibrationPattern.TcPOU
{attribute 'linkalways'} 
{attribute 'no_explicit_call' := 'This FB is a CLASS and must be accessed using methods or properties'}
{attribute 'enable_dynamic_creation'}
FUNCTION_BLOCK _ETcVnCalibrationPattern EXTENDS EnumDatatypeBase
VAR
	localData : ETcVnCalibrationPattern;
	activeData : REFERENCE TO ETcVnCalibrationPattern;
	enumBaseDatatype : _DINT(localData);
END_VAR

METHOD PRIVATE AddLocalEnumeration
VAR_INPUT
	Enumeration : T_MAXSTRING;
	Value : ETcVnCalibrationPattern;
END_VAR
AddEnumeration(Enumeration, Value);
END_METHOD

PROPERTY PUBLIC Address : PVOID
GET
Address := ADR(activeData);
END_GET
END_PROPERTY

METHOD PUBLIC ClearReference
VAR_INPUT
END_VAR
activeData REF= localData;
SetBaseDatatypeReference();
END_METHOD

METHOD PUBLIC Clone : I_Datatype
VAR
    pClone : POINTER TO _ETcVnCalibrationPattern;
END_VAR
pClone := __NEW(_ETcVnCalibrationPattern(InitialValue := Value));
Clone := pClone^;
END_METHOD

METHOD FB_init : BOOL
VAR_INPUT
	bInitRetains : BOOL; // if TRUE, the retain variables are initialized (warm start / cold start)
	bInCopyCode : BOOL;  // if TRUE, the instance afterwards gets moved into the copy code (online change)
	InitialValue : ETcVnCalibrationPattern;
END_VAR
localData := InitialValue;
AddBaseDatatype(enumBaseDatatype);
ClearReference();

AddLocalEnumeration('TCVN_CP_CIRCLES_SYM', ETcVnCalibrationPattern.TCVN_CP_CIRCLES_SYM);
AddLocalEnumeration('TCVN_CP_CIRCLES_ASYM', ETcVnCalibrationPattern.TCVN_CP_CIRCLES_ASYM);
AddLocalEnumeration('TCVN_CP_CIRCLES_ASYM_INDENT', ETcVnCalibrationPattern.TCVN_CP_CIRCLES_ASYM_INDENT);
END_METHOD

PROPERTY PUBLIC Identifier : T_MAXSTRING
GET
Identifier := 'ETcVnCalibrationPattern';
END_GET
END_PROPERTY

METHOD IsEnumeratorValueEqual : BOOL
VAR_INPUT
	Enumerator : I_KeyValueForwardEnumerator;
END_VAR
VAR
	storedValue : ETcVnCalibrationPattern;
END_VAR
IF NOT Enumerator.TryGet(storedValue) THEN
	RETURN;
END_IF

IsEnumeratorValueEqual := storedValue = activeData;
END_METHOD

METHOD PUBLIC MakeReferenceTo
VAR_INPUT
	ReferenceTarget : REFERENCE TO ETcVnCalibrationPattern;
END_VAR
activeData REF= ReferenceTarget;
SetBaseDatatypeReference();
END_METHOD

METHOD PROTECTED SetBaseDatatypeReference
VAR_INPUT
END_VAR
enumBaseDatatype.MakeReferenceTo(activeData);
END_METHOD

PROPERTY PUBLIC Size : UDINT
GET
Size := SIZEOF(activeData);
END_GET
END_PROPERTY

METHOD TryMakeReferenceTo : BOOL
VAR_INPUT
	Target : I_Datatype;
END_VAR
VAR
	targetAsEnum : I_EnumDatatype;
	pTargetData : POINTER TO ETcVnCalibrationPattern;
END_VAR
IF NOT Target.TryResolveAsEnumDatatype(targetAsEnum) THEN
	RETURN;
END_IF

IF targetAsEnum.Identifier <> Identifier THEN
	RETURN;
END_IF

pTargetData := Target.Address;
activeData REF= pTargetData^;
SetBaseDatatypeReference();
TryMakeReferenceTo := TRUE;
END_METHOD

PROPERTY PUBLIC Value : ETcVnCalibrationPattern
GET
Value := activeData;
END_GET
SET
activeData := Value;
END_SET
END_PROPERTY

END_FUNCTION_BLOCK

// ---- Enums/_ETcVnBarcodeSearchDirection.TcPOU
{attribute 'linkalways'} 
{attribute 'no_explicit_call' := 'This FB is a CLASS and must be accessed using methods or properties'}
{attribute 'enable_dynamic_creation'}
FUNCTION_BLOCK _ETcVnBarcodeSearchDirection EXTENDS EnumDatatypeBase
VAR
	localData : ETcVnBarcodeSearchDirection;
	activeData : REFERENCE TO ETcVnBarcodeSearchDirection;
	enumBaseDatatype : _UDINT(localData);
END_VAR

METHOD PRIVATE AddLocalEnumeration
VAR_INPUT
	Enumeration : T_MAXSTRING;
	Value : ETcVnBarcodeSearchDirection;
END_VAR
AddEnumeration(Enumeration, Value);
END_METHOD

PROPERTY PUBLIC Address : PVOID
GET
Address := ADR(activeData);
END_GET
END_PROPERTY

METHOD PUBLIC ClearReference
VAR_INPUT
END_VAR
activeData REF= localData;
SetBaseDatatypeReference();
END_METHOD

METHOD PUBLIC Clone : I_Datatype
VAR
    pClone : POINTER TO _ETcVnBarcodeSearchDirection;
END_VAR
pClone := __NEW(_ETcVnBarcodeSearchDirection(InitialValue := Value));
Clone := pClone^;
END_METHOD

METHOD FB_init : BOOL
VAR_INPUT
	bInitRetains : BOOL; // if TRUE, the retain variables are initialized (warm start / cold start)
	bInCopyCode : BOOL;  // if TRUE, the instance afterwards gets moved into the copy code (online change)
	InitialValue : ETcVnBarcodeSearchDirection;
END_VAR
localData := InitialValue;
AddBaseDatatype(enumBaseDatatype);
ClearReference();

AddLocalEnumeration('TCVN_BSD_ANY', ETcVnBarcodeSearchDirection.TCVN_BSD_ANY);
AddLocalEnumeration('TCVN_BSD_HORIZONTAL', ETcVnBarcodeSearchDirection.TCVN_BSD_HORIZONTAL);
AddLocalEnumeration('TCVN_BSD_VERTICAL', ETcVnBarcodeSearchDirection.TCVN_BSD_VERTICAL);
END_METHOD

PROPERTY PUBLIC Identifier : T_MAXSTRING
GET
Identifier := 'ETcVnBarcodeSearchDirection';
END_GET
END_PROPERTY

METHOD IsEnumeratorValueEqual : BOOL
VAR_INPUT
	Enumerator : I_KeyValueForwardEnumerator;
END_VAR
VAR
	storedValue : ETcVnBarcodeSearchDirection;
END_VAR
IF NOT Enumerator.TryGet(storedValue) THEN
	RETURN;
END_IF

IsEnumeratorValueEqual := storedValue = activeData;
END_METHOD

METHOD PUBLIC MakeReferenceTo
VAR_INPUT
	ReferenceTarget : REFERENCE TO ETcVnBarcodeSearchDirection;
END_VAR
activeData REF= ReferenceTarget;
SetBaseDatatypeReference();
END_METHOD

METHOD PROTECTED SetBaseDatatypeReference
VAR_INPUT
END_VAR
enumBaseDatatype.MakeReferenceTo(activeData);
END_METHOD

PROPERTY PUBLIC Size : UDINT
GET
Size := SIZEOF(activeData);
END_GET
END_PROPERTY

METHOD TryMakeReferenceTo : BOOL
VAR_INPUT
	Target : I_Datatype;
END_VAR
VAR
	targetAsEnum : I_EnumDatatype;
	pTargetData : POINTER TO ETcVnBarcodeSearchDirection;
END_VAR
IF NOT Target.TryResolveAsEnumDatatype(targetAsEnum) THEN
	RETURN;
END_IF

IF targetAsEnum.Identifier <> Identifier THEN
	RETURN;
END_IF

pTargetData := Target.Address;
activeData REF= pTargetData^;
SetBaseDatatypeReference();
TryMakeReferenceTo := TRUE;
END_METHOD

PROPERTY PUBLIC Value : ETcVnBarcodeSearchDirection
GET
Value := activeData;
END_GET
SET
activeData := Value;
END_SET
END_PROPERTY

END_FUNCTION_BLOCK

// ---- Enums/_ETcVnBarcodeType.TcPOU
{attribute 'linkalways'} 
{attribute 'no_explicit_call' := 'This FB is a CLASS and must be accessed using methods or properties'}
{attribute 'enable_dynamic_creation'}
FUNCTION_BLOCK _ETcVnBarcodeType EXTENDS EnumDatatypeBase
VAR
	localData : ETcVnBarcodeType;
	activeData : REFERENCE TO ETcVnBarcodeType;
	enumBaseDatatype : _UDINT(localData);
END_VAR

METHOD PRIVATE AddLocalEnumeration
VAR_INPUT
	Enumeration : T_MAXSTRING;
	Value : ETcVnBarcodeType;
END_VAR
AddEnumeration(Enumeration, Value);
END_METHOD

PROPERTY PUBLIC Address : PVOID
GET
Address := ADR(activeData);
END_GET
END_PROPERTY

METHOD PUBLIC ClearReference
VAR_INPUT
END_VAR
activeData REF= localData;
SetBaseDatatypeReference();
END_METHOD

METHOD PUBLIC Clone : I_Datatype
VAR
    pClone : POINTER TO _ETcVnBarcodeType;
END_VAR
pClone := __NEW(_ETcVnBarcodeType(InitialValue := Value));
Clone := pClone^;
END_METHOD

METHOD FB_init : BOOL
VAR_INPUT
	bInitRetains : BOOL; // if TRUE, the retain variables are initialized (warm start / cold start)
	bInCopyCode : BOOL;  // if TRUE, the instance afterwards gets moved into the copy code (online change)
	InitialValue : ETcVnBarcodeType;
END_VAR
localData := InitialValue;
AddBaseDatatype(enumBaseDatatype);
ClearReference();

AddLocalEnumeration('TCVN_BT_CODABAR', ETcVnBarcodeType.TCVN_BT_CODABAR);
AddLocalEnumeration('TCVN_BT_CODE39', ETcVnBarcodeType.TCVN_BT_CODE39);
AddLocalEnumeration('TCVN_BT_CODE93', ETcVnBarcodeType.TCVN_BT_CODE93);
AddLocalEnumeration('TCVN_BT_CODE128', ETcVnBarcodeType.TCVN_BT_CODE128);
AddLocalEnumeration('TCVN_BT_EAN8', ETcVnBarcodeType.TCVN_BT_EAN8);
AddLocalEnumeration('TCVN_BT_EAN13', ETcVnBarcodeType.TCVN_BT_EAN13);
AddLocalEnumeration('TCVN_BT_ITF', ETcVnBarcodeType.TCVN_BT_ITF);
AddLocalEnumeration('TCVN_BT_UPCA', ETcVnBarcodeType.TCVN_BT_UPCA);
AddLocalEnumeration('TCVN_BT_UPCE', ETcVnBarcodeType.TCVN_BT_UPCE);
AddLocalEnumeration('TCVN_BT_ANY', ETcVnBarcodeType.TCVN_BT_ANY);
AddLocalEnumeration('TCVN_BT_CODE39EXTENDED', ETcVnBarcodeType.TCVN_BT_CODE39EXTENDED);
END_METHOD

PROPERTY PUBLIC Identifier : T_MAXSTRING
GET
Identifier := 'ETcVnBarcodeType';
END_GET
END_PROPERTY

METHOD IsEnumeratorValueEqual : BOOL
VAR_INPUT
	Enumerator : I_KeyValueForwardEnumerator;
END_VAR
VAR
	storedValue : ETcVnBarcodeType;
END_VAR
IF NOT Enumerator.TryGet(storedValue) THEN
	RETURN;
END_IF

IsEnumeratorValueEqual := storedValue = activeData;
END_METHOD

METHOD PUBLIC MakeReferenceTo
VAR_INPUT
	ReferenceTarget : REFERENCE TO ETcVnBarcodeType;
END_VAR
activeData REF= ReferenceTarget;
SetBaseDatatypeReference();
END_METHOD

METHOD PROTECTED SetBaseDatatypeReference
VAR_INPUT
END_VAR
enumBaseDatatype.MakeReferenceTo(activeData);
END_METHOD

PROPERTY PUBLIC Size : UDINT
GET
Size := SIZEOF(activeData);
END_GET
END_PROPERTY

METHOD TryMakeReferenceTo : BOOL
VAR_INPUT
	Target : I_Datatype;
END_VAR
VAR
	targetAsEnum : I_EnumDatatype;
	pTargetData : POINTER TO ETcVnBarcodeType;
END_VAR
IF NOT Target.TryResolveAsEnumDatatype(targetAsEnum) THEN
	RETURN;
END_IF

IF targetAsEnum.Identifier <> Identifier THEN
	RETURN;
END_IF

pTargetData := Target.Address;
activeData REF= pTargetData^;
SetBaseDatatypeReference();
TryMakeReferenceTo := TRUE;
END_METHOD

PROPERTY PUBLIC Value : ETcVnBarcodeType
GET
Value := activeData;
END_GET
SET
activeData := Value;
END_SET
END_PROPERTY

END_FUNCTION_BLOCK

// ---- Enums/_ETcVnBlobCombination.TcPOU
{attribute 'linkalways'} 
{attribute 'no_explicit_call' := 'This FB is a CLASS and must be accessed using methods or properties'}
{attribute 'enable_dynamic_creation'}
FUNCTION_BLOCK _ETcVnBlobCombination EXTENDS EnumDatatypeBase
VAR
	localData : ETcVnBlobCombination;
	activeData : REFERENCE TO ETcVnBlobCombination;
	enumBaseDatatype : _DINT(localData);
END_VAR

METHOD PRIVATE AddLocalEnumeration
VAR_INPUT
	Enumeration : T_MAXSTRING;
	Value : ETcVnBlobCombination;
END_VAR
AddEnumeration(Enumeration, Value);
END_METHOD

PROPERTY PUBLIC Address : PVOID
GET
Address := ADR(activeData);
END_GET
END_PROPERTY

METHOD PUBLIC ClearReference
VAR_INPUT
END_VAR
activeData REF= localData;
SetBaseDatatypeReference();
END_METHOD

METHOD PUBLIC Clone : I_Datatype
VAR
    pClone : POINTER TO _ETcVnBlobCombination;
END_VAR
pClone := __NEW(_ETcVnBlobCombination(InitialValue := Value));
Clone := pClone^;
END_METHOD

METHOD FB_init : BOOL
VAR_INPUT
	bInitRetains : BOOL; // if TRUE, the retain variables are initialized (warm start / cold start)
	bInCopyCode : BOOL;  // if TRUE, the instance afterwards gets moved into the copy code (online change)
	InitialValue : ETcVnBlobCombination;
END_VAR
localData := InitialValue;
AddBaseDatatype(enumBaseDatatype);
ClearReference();

AddLocalEnumeration('TCVN_BC_SMALLEST', ETcVnBlobCombination.TCVN_BC_SMALLEST);
AddLocalEnumeration('TCVN_BC_LARGEST', ETcVnBlobCombination.TCVN_BC_LARGEST);
AddLocalEnumeration('TCVN_BC_MIN_THRESHOLD', ETcVnBlobCombination.TCVN_BC_MIN_THRESHOLD);
AddLocalEnumeration('TCVN_BC_MAX_THRESHOLD', ETcVnBlobCombination.TCVN_BC_MAX_THRESHOLD);
AddLocalEnumeration('TCVN_BC_MEDIAN_THRESHOLD', ETcVnBlobCombination.TCVN_BC_MEDIAN_THRESHOLD);
END_METHOD

PROPERTY PUBLIC Identifier : T_MAXSTRING
GET
Identifier := 'ETcVnBlobCombination';
END_GET
END_PROPERTY

METHOD IsEnumeratorValueEqual : BOOL
VAR_INPUT
	Enumerator : I_KeyValueForwardEnumerator;
END_VAR
VAR
	storedValue : ETcVnBlobCombination;
END_VAR
IF NOT Enumerator.TryGet(storedValue) THEN
	RETURN;
END_IF

IsEnumeratorValueEqual := storedValue = activeData;
END_METHOD

METHOD PUBLIC MakeReferenceTo
VAR_INPUT
	ReferenceTarget : REFERENCE TO ETcVnBlobCombination;
END_VAR
activeData REF= ReferenceTarget;
SetBaseDatatypeReference();
END_METHOD

METHOD PROTECTED SetBaseDatatypeReference
VAR_INPUT
END_VAR
enumBaseDatatype.MakeReferenceTo(activeData);
END_METHOD

PROPERTY PUBLIC Size : UDINT
GET
Size := SIZEOF(activeData);
END_GET
END_PROPERTY

METHOD TryMakeReferenceTo : BOOL
VAR_INPUT
	Target : I_Datatype;
END_VAR
VAR
	targetAsEnum : I_EnumDatatype;
	pTargetData : POINTER TO ETcVnBlobCombination;
END_VAR
IF NOT Target.TryResolveAsEnumDatatype(targetAsEnum) THEN
	RETURN;
END_IF

IF targetAsEnum.Identifier <> Identifier THEN
	RETURN;
END_IF

pTargetData := Target.Address;
activeData REF= pTargetData^;
SetBaseDatatypeReference();
TryMakeReferenceTo := TRUE;
END_METHOD

PROPERTY PUBLIC Value : ETcVnBlobCombination
GET
Value := activeData;
END_GET
SET
activeData := Value;
END_SET
END_PROPERTY

END_FUNCTION_BLOCK

// ---- Enums/_ETcVnBorderInterpolationMethod.TcPOU
{attribute 'linkalways'} 
{attribute 'no_explicit_call' := 'This FB is a CLASS and must be accessed using methods or properties'}
{attribute 'enable_dynamic_creation'}
FUNCTION_BLOCK _ETcVnBorderInterpolationMethod EXTENDS EnumDatatypeBase
VAR
	localData : ETcVnBorderInterpolationMethod;
	activeData : REFERENCE TO ETcVnBorderInterpolationMethod;
	enumBaseDatatype : _DINT(localData);
END_VAR

METHOD PRIVATE AddLocalEnumeration
VAR_INPUT
	Enumeration : T_MAXSTRING;
	Value : ETcVnBorderInterpolationMethod;
END_VAR
AddEnumeration(Enumeration, Value);
END_METHOD

PROPERTY PUBLIC Address : PVOID
GET
Address := ADR(activeData);
END_GET
END_PROPERTY

METHOD PUBLIC ClearReference
VAR_INPUT
END_VAR
activeData REF= localData;
SetBaseDatatypeReference();
END_METHOD

METHOD PUBLIC Clone : I_Datatype
VAR
    pClone : POINTER TO _ETcVnBorderInterpolationMethod;
END_VAR
pClone := __NEW(_ETcVnBorderInterpolationMethod(InitialValue := Value));
Clone := pClone^;
END_METHOD

METHOD FB_init : BOOL
VAR_INPUT
	bInitRetains : BOOL; // if TRUE, the retain variables are initialized (warm start / cold start)
	bInCopyCode : BOOL;  // if TRUE, the instance afterwards gets moved into the copy code (online change)
	InitialValue : ETcVnBorderInterpolationMethod;
END_VAR
localData := InitialValue;
AddBaseDatatype(enumBaseDatatype);
ClearReference();

AddLocalEnumeration('TCVN_BIM_CONSTANT', ETcVnBorderInterpolationMethod.TCVN_BIM_CONSTANT);
AddLocalEnumeration('TCVN_BIM_REPLICATE', ETcVnBorderInterpolationMethod.TCVN_BIM_REPLICATE);
AddLocalEnumeration('TCVN_BIM_REFLECT', ETcVnBorderInterpolationMethod.TCVN_BIM_REFLECT);
AddLocalEnumeration('TCVN_BIM_WRAP', ETcVnBorderInterpolationMethod.TCVN_BIM_WRAP);
AddLocalEnumeration('TCVN_BIM_REFLECT_101', ETcVnBorderInterpolationMethod.TCVN_BIM_REFLECT_101);
AddLocalEnumeration('TCVN_BIM_DEFAULT', ETcVnBorderInterpolationMethod.TCVN_BIM_DEFAULT);
AddLocalEnumeration('TCVN_BIM_TRANSPARENT', ETcVnBorderInterpolationMethod.TCVN_BIM_TRANSPARENT);
AddLocalEnumeration('TCVN_BIM_ISOLATED_CONSTANT', ETcVnBorderInterpolationMethod.TCVN_BIM_ISOLATED_CONSTANT);
AddLocalEnumeration('TCVN_BIM_ISOLATED_REPLICATE', ETcVnBorderInterpolationMethod.TCVN_BIM_ISOLATED_REPLICATE);
AddLocalEnumeration('TCVN_BIM_ISOLATED_REFLECT', ETcVnBorderInterpolationMethod.TCVN_BIM_ISOLATED_REFLECT);
AddLocalEnumeration('TCVN_BIM_ISOLATED_WRAP', ETcVnBorderInterpolationMethod.TCVN_BIM_ISOLATED_WRAP);
AddLocalEnumeration('TCVN_BIM_ISOLATED_REFLECT_101', ETcVnBorderInterpolationMethod.TCVN_BIM_ISOLATED_REFLECT_101);
END_METHOD

PROPERTY PUBLIC Identifier : T_MAXSTRING
GET
Identifier := 'ETcVnBorderInterpolationMethod';
END_GET
END_PROPERTY

METHOD IsEnumeratorValueEqual : BOOL
VAR_INPUT
	Enumerator : I_KeyValueForwardEnumerator;
END_VAR
VAR
	storedValue : ETcVnBorderInterpolationMethod;
END_VAR
IF NOT Enumerator.TryGet(storedValue) THEN
	RETURN;
END_IF

IsEnumeratorValueEqual := storedValue = activeData;
END_METHOD

METHOD PUBLIC MakeReferenceTo
VAR_INPUT
	ReferenceTarget : REFERENCE TO ETcVnBorderInterpolationMethod;
END_VAR
activeData REF= ReferenceTarget;
SetBaseDatatypeReference();
END_METHOD

METHOD PROTECTED SetBaseDatatypeReference
VAR_INPUT
END_VAR
enumBaseDatatype.MakeReferenceTo(activeData);
END_METHOD

PROPERTY PUBLIC Size : UDINT
GET
Size := SIZEOF(activeData);
END_GET
END_PROPERTY

METHOD TryMakeReferenceTo : BOOL
VAR_INPUT
	Target : I_Datatype;
END_VAR
VAR
	targetAsEnum : I_EnumDatatype;
	pTargetData : POINTER TO ETcVnBorderInterpolationMethod;
END_VAR
IF NOT Target.TryResolveAsEnumDatatype(targetAsEnum) THEN
	RETURN;
END_IF

IF targetAsEnum.Identifier <> Identifier THEN
	RETURN;
END_IF

pTargetData := Target.Address;
activeData REF= pTargetData^;
SetBaseDatatypeReference();
TryMakeReferenceTo := TRUE;
END_METHOD

PROPERTY PUBLIC Value : ETcVnBorderInterpolationMethod
GET
Value := activeData;
END_GET
SET
activeData := Value;
END_SET
END_PROPERTY

END_FUNCTION_BLOCK

// ---- Enums/_ETcVnCalibrationPatternOrigin.TcPOU
{attribute 'linkalways'} 
{attribute 'no_explicit_call' := 'This FB is a CLASS and must be accessed using methods or properties'}
{attribute 'enable_dynamic_creation'}
FUNCTION_BLOCK _ETcVnCalibrationPatternOrigin EXTENDS EnumDatatypeBase
VAR
	localData : ETcVnCalibrationPatternOrigin;
	activeData : REFERENCE TO ETcVnCalibrationPatternOrigin;
	enumBaseDatatype : _DINT(localData);
END_VAR

METHOD PRIVATE AddLocalEnumeration
VAR_INPUT
	Enumeration : T_MAXSTRING;
	Value : ETcVnCalibrationPatternOrigin;
END_VAR
AddEnumeration(Enumeration, Value);
END_METHOD

PROPERTY PUBLIC Address : PVOID
GET
Address := ADR(activeData);
END_GET
END_PROPERTY

METHOD PUBLIC ClearReference
VAR_INPUT
END_VAR
activeData REF= localData;
SetBaseDatatypeReference();
END_METHOD

METHOD PUBLIC Clone : I_Datatype
VAR
    pClone : POINTER TO _ETcVnCalibrationPatternOrigin;
END_VAR
pClone := __NEW(_ETcVnCalibrationPatternOrigin(InitialValue := Value));
Clone := pClone^;
END_METHOD

METHOD FB_init : BOOL
VAR_INPUT
	bInitRetains : BOOL; // if TRUE, the retain variables are initialized (warm start / cold start)
	bInCopyCode : BOOL;  // if TRUE, the instance afterwards gets moved into the copy code (online change)
	InitialValue : ETcVnCalibrationPatternOrigin;
END_VAR
localData := InitialValue;
AddBaseDatatype(enumBaseDatatype);
ClearReference();

AddLocalEnumeration('TCVN_CPO_TOPLEFT', ETcVnCalibrationPatternOrigin.TCVN_CPO_TOPLEFT);
AddLocalEnumeration('TCVN_CPO_TOPCENTER', ETcVnCalibrationPatternOrigin.TCVN_CPO_TOPCENTER);
AddLocalEnumeration('TCVN_CPO_TOPRIGHT', ETcVnCalibrationPatternOrigin.TCVN_CPO_TOPRIGHT);
AddLocalEnumeration('TCVN_CPO_CENTERLEFT', ETcVnCalibrationPatternOrigin.TCVN_CPO_CENTERLEFT);
AddLocalEnumeration('TCVN_CPO_CENTER', ETcVnCalibrationPatternOrigin.TCVN_CPO_CENTER);
AddLocalEnumeration('TCVN_CPO_CENTERRIGHT', ETcVnCalibrationPatternOrigin.TCVN_CPO_CENTERRIGHT);
AddLocalEnumeration('TCVN_CPO_BOTTOMLEFT', ETcVnCalibrationPatternOrigin.TCVN_CPO_BOTTOMLEFT);
AddLocalEnumeration('TCVN_CPO_BOTTOMCENTER', ETcVnCalibrationPatternOrigin.TCVN_CPO_BOTTOMCENTER);
AddLocalEnumeration('TCVN_CPO_BOTTOMRIGHT', ETcVnCalibrationPatternOrigin.TCVN_CPO_BOTTOMRIGHT);
END_METHOD

PROPERTY PUBLIC Identifier : T_MAXSTRING
GET
Identifier := 'ETcVnCalibrationPatternOrigin';
END_GET
END_PROPERTY

METHOD IsEnumeratorValueEqual : BOOL
VAR_INPUT
	Enumerator : I_KeyValueForwardEnumerator;
END_VAR
VAR
	storedValue : ETcVnCalibrationPatternOrigin;
END_VAR
IF NOT Enumerator.TryGet(storedValue) THEN
	RETURN;
END_IF

IsEnumeratorValueEqual := storedValue = activeData;
END_METHOD

METHOD PUBLIC MakeReferenceTo
VAR_INPUT
	ReferenceTarget : REFERENCE TO ETcVnCalibrationPatternOrigin;
END_VAR
activeData REF= ReferenceTarget;
SetBaseDatatypeReference();
END_METHOD

METHOD PROTECTED SetBaseDatatypeReference
VAR_INPUT
END_VAR
enumBaseDatatype.MakeReferenceTo(activeData);
END_METHOD

PROPERTY PUBLIC Size : UDINT
GET
Size := SIZEOF(activeData);
END_GET
END_PROPERTY

METHOD TryMakeReferenceTo : BOOL
VAR_INPUT
	Target : I_Datatype;
END_VAR
VAR
	targetAsEnum : I_EnumDatatype;
	pTargetData : POINTER TO ETcVnCalibrationPatternOrigin;
END_VAR
IF NOT Target.TryResolveAsEnumDatatype(targetAsEnum) THEN
	RETURN;
END_IF

IF targetAsEnum.Identifier <> Identifier THEN
	RETURN;
END_IF

pTargetData := Target.Address;
activeData REF= pTargetData^;
SetBaseDatatypeReference();
TryMakeReferenceTo := TRUE;
END_METHOD

PROPERTY PUBLIC Value : ETcVnCalibrationPatternOrigin
GET
Value := activeData;
END_GET
SET
activeData := Value;
END_SET
END_PROPERTY

END_FUNCTION_BLOCK

// ---- Enums/_ETcVnCameraState.TcPOU
{attribute 'linkalways'} 
{attribute 'no_explicit_call' := 'This FB is a CLASS and must be accessed using methods or properties'}
{attribute 'enable_dynamic_creation'}
FUNCTION_BLOCK _ETcVnCameraState EXTENDS EnumDatatypeBase
VAR
	localData : ETcVnCameraState;
	activeData : REFERENCE TO ETcVnCameraState;
	enumBaseDatatype : _DINT(localData);
END_VAR

METHOD PRIVATE AddLocalEnumeration
VAR_INPUT
	Enumeration : T_MAXSTRING;
	Value : ETcVnCameraState;
END_VAR
AddEnumeration(Enumeration, Value);
END_METHOD

PROPERTY PUBLIC Address : PVOID
GET
Address := ADR(activeData);
END_GET
END_PROPERTY

METHOD PUBLIC ClearReference
VAR_INPUT
END_VAR
activeData REF= localData;
SetBaseDatatypeReference();
END_METHOD

METHOD PUBLIC Clone : I_Datatype
VAR
    pClone : POINTER TO _ETcVnCameraState;
END_VAR
pClone := __NEW(_ETcVnCameraState(InitialValue := Value));
Clone := pClone^;
END_METHOD

METHOD FB_init : BOOL
VAR_INPUT
	bInitRetains : BOOL; // if TRUE, the retain variables are initialized (warm start / cold start)
	bInCopyCode : BOOL;  // if TRUE, the instance afterwards gets moved into the copy code (online change)
	InitialValue : ETcVnCameraState;
END_VAR
localData := InitialValue;
AddBaseDatatype(enumBaseDatatype);
ClearReference();

AddLocalEnumeration('TCVN_CS_ERROR', ETcVnCameraState.TCVN_CS_ERROR);
AddLocalEnumeration('TCVN_CS_INITIAL', ETcVnCameraState.TCVN_CS_INITIAL);
AddLocalEnumeration('TCVN_CS_INITIALIZING', ETcVnCameraState.TCVN_CS_INITIALIZING);
AddLocalEnumeration('TCVN_CS_INITIALIZED', ETcVnCameraState.TCVN_CS_INITIALIZED);
AddLocalEnumeration('TCVN_CS_OPENING', ETcVnCameraState.TCVN_CS_OPENING);
AddLocalEnumeration('TCVN_CS_OPENED', ETcVnCameraState.TCVN_CS_OPENED);
AddLocalEnumeration('TCVN_CS_STARTACQUISITION', ETcVnCameraState.TCVN_CS_STARTACQUISITION);
AddLocalEnumeration('TCVN_CS_ACQUIRING', ETcVnCameraState.TCVN_CS_ACQUIRING);
AddLocalEnumeration('TCVN_CS_STOPACQUISITION', ETcVnCameraState.TCVN_CS_STOPACQUISITION);
AddLocalEnumeration('TCVN_CS_RESETTINGFEATURES', ETcVnCameraState.TCVN_CS_RESETTINGFEATURES);
AddLocalEnumeration('TCVN_CS_TRIGGERING', ETcVnCameraState.TCVN_CS_TRIGGERING);
AddLocalEnumeration('TCVN_CS_CLOSING', ETcVnCameraState.TCVN_CS_CLOSING);
END_METHOD

PROPERTY PUBLIC Identifier : T_MAXSTRING
GET
Identifier := 'ETcVnCameraState';
END_GET
END_PROPERTY

METHOD IsEnumeratorValueEqual : BOOL
VAR_INPUT
	Enumerator : I_KeyValueForwardEnumerator;
END_VAR
VAR
	storedValue : ETcVnCameraState;
END_VAR
IF NOT Enumerator.TryGet(storedValue) THEN
	RETURN;
END_IF

IsEnumeratorValueEqual := storedValue = activeData;
END_METHOD

METHOD PUBLIC MakeReferenceTo
VAR_INPUT
	ReferenceTarget : REFERENCE TO ETcVnCalibrationPatternOrigin;
END_VAR
activeData REF= ReferenceTarget;
SetBaseDatatypeReference();
END_METHOD

METHOD PROTECTED SetBaseDatatypeReference
VAR_INPUT
END_VAR
enumBaseDatatype.MakeReferenceTo(activeData);
END_METHOD

PROPERTY PUBLIC Size : UDINT
GET
Size := SIZEOF(activeData);
END_GET
END_PROPERTY

METHOD TryMakeReferenceTo : BOOL
VAR_INPUT
	Target : I_Datatype;
END_VAR
VAR
	targetAsEnum : I_EnumDatatype;
	pTargetData : POINTER TO ETcVnCameraState;
END_VAR
IF NOT Target.TryResolveAsEnumDatatype(targetAsEnum) THEN
	RETURN;
END_IF

IF targetAsEnum.Identifier <> Identifier THEN
	RETURN;
END_IF

pTargetData := Target.Address;
activeData REF= pTargetData^;
SetBaseDatatypeReference();
TryMakeReferenceTo := TRUE;
END_METHOD

PROPERTY PUBLIC Value : ETcVnCameraState
GET
Value := activeData;
END_GET
SET
activeData := Value;
END_SET
END_PROPERTY

END_FUNCTION_BLOCK

// ---- Enums/_ETcVnClusteringAlgorithm.TcPOU
{attribute 'linkalways'} 
{attribute 'no_explicit_call' := 'This FB is a CLASS and must be accessed using methods or properties'}
{attribute 'enable_dynamic_creation'}
FUNCTION_BLOCK _ETcVnClusteringAlgorithm EXTENDS EnumDatatypeBase
VAR
	localData : ETcVnClusteringAlgorithm;
	activeData : REFERENCE TO ETcVnClusteringAlgorithm;
	enumBaseDatatype : _DINT(localData);
END_VAR

METHOD PRIVATE AddLocalEnumeration
VAR_INPUT
	Enumeration : T_MAXSTRING;
	Value : ETcVnClusteringAlgorithm;
END_VAR
AddEnumeration(Enumeration, Value);
END_METHOD

PROPERTY PUBLIC Address : PVOID
GET
Address := ADR(activeData);
END_GET
END_PROPERTY

METHOD PUBLIC ClearReference
VAR_INPUT
END_VAR
activeData REF= localData;
SetBaseDatatypeReference();
END_METHOD

METHOD PUBLIC Clone : I_Datatype
VAR
    pClone : POINTER TO _ETcVnClusteringAlgorithm;
END_VAR
pClone := __NEW(_ETcVnClusteringAlgorithm(InitialValue := Value));
Clone := pClone^;
END_METHOD

METHOD FB_init : BOOL
VAR_INPUT
	bInitRetains : BOOL; // if TRUE, the retain variables are initialized (warm start / cold start)
	bInCopyCode : BOOL;  // if TRUE, the instance afterwards gets moved into the copy code (online change)
	InitialValue : ETcVnClusteringAlgorithm;
END_VAR
localData := InitialValue;
AddBaseDatatype(enumBaseDatatype);
ClearReference();

AddLocalEnumeration('TCVN_CA_KMEANSPP', ETcVnClusteringAlgorithm.TCVN_CA_KMEANSPP);
AddLocalEnumeration('TCVN_CA_LBG', ETcVnClusteringAlgorithm.TCVN_CA_LBG);
END_METHOD

PROPERTY PUBLIC Identifier : T_MAXSTRING
GET
Identifier := 'ETcVnClusteringAlgorithm';
END_GET
END_PROPERTY

METHOD IsEnumeratorValueEqual : BOOL
VAR_INPUT
	Enumerator : I_KeyValueForwardEnumerator;
END_VAR
VAR
	storedValue : ETcVnClusteringAlgorithm;
END_VAR
IF NOT Enumerator.TryGet(storedValue) THEN
	RETURN;
END_IF

IsEnumeratorValueEqual := storedValue = activeData;
END_METHOD

METHOD PUBLIC MakeReferenceTo
VAR_INPUT
	ReferenceTarget : REFERENCE TO ETcVnCalibrationPatternOrigin;
END_VAR
activeData REF= ReferenceTarget;
SetBaseDatatypeReference();
END_METHOD

METHOD PROTECTED SetBaseDatatypeReference
VAR_INPUT
END_VAR
enumBaseDatatype.MakeReferenceTo(activeData);
END_METHOD

PROPERTY PUBLIC Size : UDINT
GET
Size := SIZEOF(activeData);
END_GET
END_PROPERTY

METHOD TryMakeReferenceTo : BOOL
VAR_INPUT
	Target : I_Datatype;
END_VAR
VAR
	targetAsEnum : I_EnumDatatype;
	pTargetData : POINTER TO ETcVnClusteringAlgorithm;
END_VAR
IF NOT Target.TryResolveAsEnumDatatype(targetAsEnum) THEN
	RETURN;
END_IF

IF targetAsEnum.Identifier <> Identifier THEN
	RETURN;
END_IF

pTargetData := Target.Address;
activeData REF= pTargetData^;
SetBaseDatatypeReference();
TryMakeReferenceTo := TRUE;
END_METHOD

PROPERTY PUBLIC Value : ETcVnClusteringAlgorithm
GET
Value := activeData;
END_GET
SET
activeData := Value;
END_SET
END_PROPERTY

END_FUNCTION_BLOCK

// ---- Enums/_ETcVnColorMap.TcPOU
{attribute 'linkalways'} 
{attribute 'no_explicit_call' := 'This FB is a CLASS and must be accessed using methods or properties'}
{attribute 'enable_dynamic_creation'}
FUNCTION_BLOCK _ETcVnColorMap EXTENDS EnumDatatypeBase
VAR
	localData : ETcVnColorMap;
	activeData : REFERENCE TO ETcVnColorMap;
	enumBaseDatatype : _DINT(localData);
END_VAR

METHOD PRIVATE AddLocalEnumeration
VAR_INPUT
	Enumeration : T_MAXSTRING;
	Value : ETcVnColorMap;
END_VAR
AddEnumeration(Enumeration, Value);
END_METHOD

PROPERTY PUBLIC Address : PVOID
GET
Address := ADR(activeData);
END_GET
END_PROPERTY

METHOD PUBLIC ClearReference
VAR_INPUT
END_VAR
activeData REF= localData;
SetBaseDatatypeReference();
END_METHOD

METHOD PUBLIC Clone : I_Datatype
VAR
    pClone : POINTER TO _ETcVnColorMap;
END_VAR
pClone := __NEW(_ETcVnColorMap(InitialValue := Value));
Clone := pClone^;
END_METHOD

METHOD FB_init : BOOL
VAR_INPUT
	bInitRetains : BOOL; // if TRUE, the retain variables are initialized (warm start / cold start)
	bInCopyCode : BOOL;  // if TRUE, the instance afterwards gets moved into the copy code (online change)
	InitialValue : ETcVnColorMap;
END_VAR
localData := InitialValue;
AddBaseDatatype(enumBaseDatatype);
ClearReference();

AddLocalEnumeration('TCVN_CM_AUTUMN', ETcVnColorMap.TCVN_CM_AUTUMN);
AddLocalEnumeration('TCVN_CM_BONE', ETcVnColorMap.TCVN_CM_BONE);
AddLocalEnumeration('TCVN_CM_JET', ETcVnColorMap.TCVN_CM_JET);
AddLocalEnumeration('TCVN_CM_WINTER', ETcVnColorMap.TCVN_CM_WINTER);
AddLocalEnumeration('TCVN_CM_RAINBOW', ETcVnColorMap.TCVN_CM_RAINBOW);
AddLocalEnumeration('TCVN_CM_OCEAN', ETcVnColorMap.TCVN_CM_OCEAN);
AddLocalEnumeration('TCVN_CM_SUMMER', ETcVnColorMap.TCVN_CM_SUMMER);
AddLocalEnumeration('TCVN_CM_SPRING', ETcVnColorMap.TCVN_CM_SPRING);
AddLocalEnumeration('TCVN_CM_COOL', ETcVnColorMap.TCVN_CM_COOL);
AddLocalEnumeration('TCVN_CM_HSV', ETcVnColorMap.TCVN_CM_HSV);
AddLocalEnumeration('TCVN_CM_PINK', ETcVnColorMap.TCVN_CM_PINK);
AddLocalEnumeration('TCVN_CM_HOT', ETcVnColorMap.TCVN_CM_HOT);
AddLocalEnumeration('TCVN_CM_PARULA', ETcVnColorMap.TCVN_CM_PARULA);
AddLocalEnumeration('TCVN_CM_MAGMA', ETcVnColorMap.TCVN_CM_MAGMA);
AddLocalEnumeration('TCVN_CM_INFERNO', ETcVnColorMap.TCVN_CM_INFERNO);
AddLocalEnumeration('TCVN_CM_PLASMA', ETcVnColorMap.TCVN_CM_PLASMA);
AddLocalEnumeration('TCVN_CM_VIRIDIS', ETcVnColorMap.TCVN_CM_VIRIDIS);
AddLocalEnumeration('TCVN_CM_CIVIDIS', ETcVnColorMap.TCVN_CM_CIVIDIS);
AddLocalEnumeration('TCVN_CM_TWILIGHT', ETcVnColorMap.TCVN_CM_TWILIGHT);
AddLocalEnumeration('TCVN_CM_TWILIGHT_SHIFTED', ETcVnColorMap.TCVN_CM_TWILIGHT_SHIFTED);
AddLocalEnumeration('TCVN_CM_TURBO', ETcVnColorMap.TCVN_CM_TURBO);
END_METHOD

PROPERTY PUBLIC Identifier : T_MAXSTRING
GET
Identifier := 'ETcVnColorMap';
END_GET
END_PROPERTY

METHOD IsEnumeratorValueEqual : BOOL
VAR_INPUT
	Enumerator : I_KeyValueForwardEnumerator;
END_VAR
VAR
	storedValue : ETcVnColorMap;
END_VAR
IF NOT Enumerator.TryGet(storedValue) THEN
	RETURN;
END_IF

IsEnumeratorValueEqual := storedValue = activeData;
END_METHOD

METHOD PUBLIC MakeReferenceTo
VAR_INPUT
	ReferenceTarget : REFERENCE TO ETcVnCalibrationPatternOrigin;
END_VAR
activeData REF= ReferenceTarget;
SetBaseDatatypeReference();
END_METHOD

METHOD PROTECTED SetBaseDatatypeReference
VAR_INPUT
END_VAR
enumBaseDatatype.MakeReferenceTo(activeData);
END_METHOD

PROPERTY PUBLIC Size : UDINT
GET
Size := SIZEOF(activeData);
END_GET
END_PROPERTY

METHOD TryMakeReferenceTo : BOOL
VAR_INPUT
	Target : I_Datatype;
END_VAR
VAR
	targetAsEnum : I_EnumDatatype;
	pTargetData : POINTER TO ETcVnColorMap;
END_VAR
IF NOT Target.TryResolveAsEnumDatatype(targetAsEnum) THEN
	RETURN;
END_IF

IF targetAsEnum.Identifier <> Identifier THEN
	RETURN;
END_IF

pTargetData := Target.Address;
activeData REF= pTargetData^;
SetBaseDatatypeReference();
TryMakeReferenceTo := TRUE;
END_METHOD

PROPERTY PUBLIC Value : ETcVnColorMap
GET
Value := activeData;
END_GET
SET
activeData := Value;
END_SET
END_PROPERTY

END_FUNCTION_BLOCK

// ---- Enums/_ETcVnColorSpaceTransform.TcPOU
{attribute 'linkalways'} 
{attribute 'no_explicit_call' := 'This FB is a CLASS and must be accessed using methods or properties'}
{attribute 'enable_dynamic_creation'}
FUNCTION_BLOCK _ETcVnColorSpaceTransform EXTENDS EnumDatatypeBase
VAR
	localData : ETcVnColorSpaceTransform;
	activeData : REFERENCE TO ETcVnColorSpaceTransform;
	enumBaseDatatype : _DINT(localData);
END_VAR

METHOD PRIVATE AddLocalEnumeration
VAR_INPUT
	Enumeration : T_MAXSTRING;
	Value : ETcVnColorSpaceTransform;
END_VAR
AddEnumeration(Enumeration, Value);
END_METHOD

PROPERTY PUBLIC Address : PVOID
GET
Address := ADR(activeData);
END_GET
END_PROPERTY

METHOD PUBLIC ClearReference
VAR_INPUT
END_VAR
activeData REF= localData;
SetBaseDatatypeReference();
END_METHOD

METHOD PUBLIC Clone : I_Datatype
VAR
    pClone : POINTER TO _ETcVnColorSpaceTransform;
END_VAR
pClone := __NEW(_ETcVnColorSpaceTransform(InitialValue := Value));
Clone := pClone^;
END_METHOD

METHOD FB_init : BOOL
VAR_INPUT
	bInitRetains : BOOL; // if TRUE, the retain variables are initialized (warm start / cold start)
	bInCopyCode : BOOL;  // if TRUE, the instance afterwards gets moved into the copy code (online change)
	InitialValue : ETcVnColorSpaceTransform;
END_VAR
localData := InitialValue;
AddBaseDatatype(enumBaseDatatype);
ClearReference();

AddLocalEnumeration('TCVN_CST_BGR_TO_BGRA', ETcVnColorSpaceTransform.TCVN_CST_BGR_TO_BGRA);
AddLocalEnumeration('TCVN_CST_RGB_TO_RGBA', ETcVnColorSpaceTransform.TCVN_CST_RGB_TO_RGBA);
AddLocalEnumeration('TCVN_CST_BGRA_TO_BGR', ETcVnColorSpaceTransform.TCVN_CST_BGRA_TO_BGR);
AddLocalEnumeration('TCVN_CST_RGBA_TO_RGB', ETcVnColorSpaceTransform.TCVN_CST_RGBA_TO_RGB);
AddLocalEnumeration('TCVN_CST_BGR_TO_RGBA', ETcVnColorSpaceTransform.TCVN_CST_BGR_TO_RGBA);
AddLocalEnumeration('TCVN_CST_RGB_TO_BGRA', ETcVnColorSpaceTransform.TCVN_CST_RGB_TO_BGRA);
AddLocalEnumeration('TCVN_CST_BGRA_TO_RGB', ETcVnColorSpaceTransform.TCVN_CST_BGRA_TO_RGB);
AddLocalEnumeration('TCVN_CST_RGBA_TO_BGR', ETcVnColorSpaceTransform.TCVN_CST_RGBA_TO_BGR);
AddLocalEnumeration('TCVN_CST_BGR_TO_RGB', ETcVnColorSpaceTransform.TCVN_CST_BGR_TO_RGB);
AddLocalEnumeration('TCVN_CST_RGB_TO_BGR', ETcVnColorSpaceTransform.TCVN_CST_RGB_TO_BGR);
AddLocalEnumeration('TCVN_CST_BGRA_TO_RGBA', ETcVnColorSpaceTransform.TCVN_CST_BGRA_TO_RGBA);
AddLocalEnumeration('TCVN_CST_RGBA_TO_BGRA', ETcVnColorSpaceTransform.TCVN_CST_RGBA_TO_BGRA);
AddLocalEnumeration('TCVN_CST_BGR_TO_GRAY', ETcVnColorSpaceTransform.TCVN_CST_BGR_TO_GRAY);
AddLocalEnumeration('TCVN_CST_RGB_TO_GRAY', ETcVnColorSpaceTransform.TCVN_CST_RGB_TO_GRAY);
AddLocalEnumeration('TCVN_CST_GRAY_TO_BGR', ETcVnColorSpaceTransform.TCVN_CST_GRAY_TO_BGR);
AddLocalEnumeration('TCVN_CST_GRAY_TO_RGB', ETcVnColorSpaceTransform.TCVN_CST_GRAY_TO_RGB);
AddLocalEnumeration('TCVN_CST_GRAY_TO_BGRA', ETcVnColorSpaceTransform.TCVN_CST_GRAY_TO_BGRA);
AddLocalEnumeration('TCVN_CST_GRAY_TO_RGBA', ETcVnColorSpaceTransform.TCVN_CST_GRAY_TO_RGBA);
AddLocalEnumeration('TCVN_CST_BGRA_TO_GRAY', ETcVnColorSpaceTransform.TCVN_CST_BGRA_TO_GRAY);
AddLocalEnumeration('TCVN_CST_RGBA_TO_GRAY', ETcVnColorSpaceTransform.TCVN_CST_RGBA_TO_GRAY);
AddLocalEnumeration('TCVN_CST_RGB_TO_BGR_565', ETcVnColorSpaceTransform.TCVN_CST_RGB_TO_BGR_565);
AddLocalEnumeration('TCVN_CST_BGR_TO_BGR_565', ETcVnColorSpaceTransform.TCVN_CST_BGR_TO_BGR_565);
AddLocalEnumeration('TCVN_CST_BGR_565_TO_RGB', ETcVnColorSpaceTransform.TCVN_CST_BGR_565_TO_RGB);
AddLocalEnumeration('TCVN_CST_BGR_565_TO_BGR', ETcVnColorSpaceTransform.TCVN_CST_BGR_565_TO_BGR);
AddLocalEnumeration('TCVN_CST_RGBA_TO_BGR_565', ETcVnColorSpaceTransform.TCVN_CST_RGBA_TO_BGR_565);
AddLocalEnumeration('TCVN_CST_BGRA_TO_BGR_565', ETcVnColorSpaceTransform.TCVN_CST_BGRA_TO_BGR_565);
AddLocalEnumeration('TCVN_CST_BGR_565_TO_RGBA', ETcVnColorSpaceTransform.TCVN_CST_BGR_565_TO_RGBA);
AddLocalEnumeration('TCVN_CST_BGR_565_TO_BGRA', ETcVnColorSpaceTransform.TCVN_CST_BGR_565_TO_BGRA);
AddLocalEnumeration('TCVN_CST_GRAY_TO_BGR_565', ETcVnColorSpaceTransform.TCVN_CST_GRAY_TO_BGR_565);
AddLocalEnumeration('TCVN_CST_BGR_565_TO_GRAY', ETcVnColorSpaceTransform.TCVN_CST_BGR_565_TO_GRAY);
AddLocalEnumeration('TCVN_CST_RGB_TO_BGR_555', ETcVnColorSpaceTransform.TCVN_CST_RGB_TO_BGR_555);
AddLocalEnumeration('TCVN_CST_BGR_TO_BGR_555', ETcVnColorSpaceTransform.TCVN_CST_BGR_TO_BGR_555);
AddLocalEnumeration('TCVN_CST_BGR_555_TO_RGB', ETcVnColorSpaceTransform.TCVN_CST_BGR_555_TO_RGB);
AddLocalEnumeration('TCVN_CST_BGR_555_TO_BGR', ETcVnColorSpaceTransform.TCVN_CST_BGR_555_TO_BGR);
AddLocalEnumeration('TCVN_CST_RGBA_TO_BGR_555', ETcVnColorSpaceTransform.TCVN_CST_RGBA_TO_BGR_555);
AddLocalEnumeration('TCVN_CST_BGRA_TO_BGR_555', ETcVnColorSpaceTransform.TCVN_CST_BGRA_TO_BGR_555);
AddLocalEnumeration('TCVN_CST_BGR_555_TO_RGBA', ETcVnColorSpaceTransform.TCVN_CST_BGR_555_TO_RGBA);
AddLocalEnumeration('TCVN_CST_BGR_555_TO_BGRA', ETcVnColorSpaceTransform.TCVN_CST_BGR_555_TO_BGRA);
AddLocalEnumeration('TCVN_CST_GRAY_TO_BGR_555', ETcVnColorSpaceTransform.TCVN_CST_GRAY_TO_BGR_555);
AddLocalEnumeration('TCVN_CST_BGR_555_TO_GRAY', ETcVnColorSpaceTransform.TCVN_CST_BGR_555_TO_GRAY);
AddLocalEnumeration('TCVN_CST_BGR_TO_XYZ', ETcVnColorSpaceTransform.TCVN_CST_BGR_TO_XYZ);
AddLocalEnumeration('TCVN_CST_RGB_TO_XYZ', ETcVnColorSpaceTransform.TCVN_CST_RGB_TO_XYZ);
AddLocalEnumeration('TCVN_CST_XYZ_TO_BGR', ETcVnColorSpaceTransform.TCVN_CST_XYZ_TO_BGR);
AddLocalEnumeration('TCVN_CST_XYZ_TO_RGB', ETcVnColorSpaceTransform.TCVN_CST_XYZ_TO_RGB);
AddLocalEnumeration('TCVN_CST_BGR_TO_YCRCB', ETcVnColorSpaceTransform.TCVN_CST_BGR_TO_YCRCB);
AddLocalEnumeration('TCVN_CST_RGB_TO_YCRCB', ETcVnColorSpaceTransform.TCVN_CST_RGB_TO_YCRCB);
AddLocalEnumeration('TCVN_CST_YCRCB_TO_BGR', ETcVnColorSpaceTransform.TCVN_CST_YCRCB_TO_BGR);
AddLocalEnumeration('TCVN_CST_YCRCB_TO_RGB', ETcVnColorSpaceTransform.TCVN_CST_YCRCB_TO_RGB);
AddLocalEnumeration('TCVN_CST_BGR_TO_HSV', ETcVnColorSpaceTransform.TCVN_CST_BGR_TO_HSV);
AddLocalEnumeration('TCVN_CST_RGB_TO_HSV', ETcVnColorSpaceTransform.TCVN_CST_RGB_TO_HSV);
AddLocalEnumeration('TCVN_CST_BGR_TO_LAB', ETcVnColorSpaceTransform.TCVN_CST_BGR_TO_LAB);
AddLocalEnumeration('TCVN_CST_RGB_TO_LAB', ETcVnColorSpaceTransform.TCVN_CST_RGB_TO_LAB);
AddLocalEnumeration('TCVN_CST_BAYER_RG_TO_BGR', ETcVnColorSpaceTransform.TCVN_CST_BAYER_RG_TO_BGR);
AddLocalEnumeration('TCVN_CST_BAYER_BG_TO_RGB', ETcVnColorSpaceTransform.TCVN_CST_BAYER_BG_TO_RGB);
AddLocalEnumeration('TCVN_CST_BAYER_GR_TO_BGR', ETcVnColorSpaceTransform.TCVN_CST_BAYER_GR_TO_BGR);
AddLocalEnumeration('TCVN_CST_BAYER_GB_TO_RGB', ETcVnColorSpaceTransform.TCVN_CST_BAYER_GB_TO_RGB);
AddLocalEnumeration('TCVN_CST_BAYER_BG_TO_BGR', ETcVnColorSpaceTransform.TCVN_CST_BAYER_BG_TO_BGR);
AddLocalEnumeration('TCVN_CST_BAYER_RG_TO_RGB', ETcVnColorSpaceTransform.TCVN_CST_BAYER_RG_TO_RGB);
AddLocalEnumeration('TCVN_CST_BAYER_GB_TO_BGR', ETcVnColorSpaceTransform.TCVN_CST_BAYER_GB_TO_BGR);
AddLocalEnumeration('TCVN_CST_BAYER_GR_TO_RGB', ETcVnColorSpaceTransform.TCVN_CST_BAYER_GR_TO_RGB);
AddLocalEnumeration('TCVN_CST_BGR_TO_LUV', ETcVnColorSpaceTransform.TCVN_CST_BGR_TO_LUV);
AddLocalEnumeration('TCVN_CST_RGB_TO_LUV', ETcVnColorSpaceTransform.TCVN_CST_RGB_TO_LUV);
AddLocalEnumeration('TCVN_CST_BGR_TO_HLS', ETcVnColorSpaceTransform.TCVN_CST_BGR_TO_HLS);
AddLocalEnumeration('TCVN_CST_RGB_TO_HLS', ETcVnColorSpaceTransform.TCVN_CST_RGB_TO_HLS);
AddLocalEnumeration('TCVN_CST_HSV_TO_BGR', ETcVnColorSpaceTransform.TCVN_CST_HSV_TO_BGR);
AddLocalEnumeration('TCVN_CST_HSV_TO_RGB', ETcVnColorSpaceTransform.TCVN_CST_HSV_TO_RGB);
AddLocalEnumeration('TCVN_CST_LAB_TO_BGR', ETcVnColorSpaceTransform.TCVN_CST_LAB_TO_BGR);
AddLocalEnumeration('TCVN_CST_LAB_TO_RGB', ETcVnColorSpaceTransform.TCVN_CST_LAB_TO_RGB);
AddLocalEnumeration('TCVN_CST_LUV_TO_BGR', ETcVnColorSpaceTransform.TCVN_CST_LUV_TO_BGR);
AddLocalEnumeration('TCVN_CST_LUV_TO_RGB', ETcVnColorSpaceTransform.TCVN_CST_LUV_TO_RGB);
AddLocalEnumeration('TCVN_CST_HLS_TO_BGR', ETcVnColorSpaceTransform.TCVN_CST_HLS_TO_BGR);
AddLocalEnumeration('TCVN_CST_HLS_TO_RGB', ETcVnColorSpaceTransform.TCVN_CST_HLS_TO_RGB);
AddLocalEnumeration('TCVN_CST_BAYER_RG_TO_BGR_VNG', ETcVnColorSpaceTransform.TCVN_CST_BAYER_RG_TO_BGR_VNG);
AddLocalEnumeration('TCVN_CST_BAYER_GR_TO_BGR_VNG', ETcVnColorSpaceTransform.TCVN_CST_BAYER_GR_TO_BGR_VNG);
AddLocalEnumeration('TCVN_CST_BAYER_BG_TO_BGR_VNG', ETcVnColorSpaceTransform.TCVN_CST_BAYER_BG_TO_BGR_VNG);
AddLocalEnumeration('TCVN_CST_BAYER_GB_TO_BGR_VNG', ETcVnColorSpaceTransform.TCVN_CST_BAYER_GB_TO_BGR_VNG);
AddLocalEnumeration('TCVN_CST_BAYER_RG_TO_RGB_VNG', ETcVnColorSpaceTransform.TCVN_CST_BAYER_RG_TO_RGB_VNG);
AddLocalEnumeration('TCVN_CST_BAYER_GR_TO_RGB_VNG', ETcVnColorSpaceTransform.TCVN_CST_BAYER_GR_TO_RGB_VNG);
AddLocalEnumeration('TCVN_CST_BAYER_BG_TO_RGB_VNG', ETcVnColorSpaceTransform.TCVN_CST_BAYER_BG_TO_RGB_VNG);
AddLocalEnumeration('TCVN_CST_BAYER_GB_TO_RGB_VNG', ETcVnColorSpaceTransform.TCVN_CST_BAYER_GB_TO_RGB_VNG);
AddLocalEnumeration('TCVN_CST_BGR_TO_HSV_FULL', ETcVnColorSpaceTransform.TCVN_CST_BGR_TO_HSV_FULL);
AddLocalEnumeration('TCVN_CST_RGB_TO_HSV_FULL', ETcVnColorSpaceTransform.TCVN_CST_RGB_TO_HSV_FULL);
AddLocalEnumeration('TCVN_CST_BGR_TO_HLS_FULL', ETcVnColorSpaceTransform.TCVN_CST_BGR_TO_HLS_FULL);
AddLocalEnumeration('TCVN_CST_RGB_TO_HLS_FULL', ETcVnColorSpaceTransform.TCVN_CST_RGB_TO_HLS_FULL);
AddLocalEnumeration('TCVN_CST_HSV_TO_BGR_FULL', ETcVnColorSpaceTransform.TCVN_CST_HSV_TO_BGR_FULL);
AddLocalEnumeration('TCVN_CST_HSV_TO_RGB_FULL', ETcVnColorSpaceTransform.TCVN_CST_HSV_TO_RGB_FULL);
AddLocalEnumeration('TCVN_CST_HLS_TO_BGR_FULL', ETcVnColorSpaceTransform.TCVN_CST_HLS_TO_BGR_FULL);
AddLocalEnumeration('TCVN_CST_HLS_TO_RGB_FULL', ETcVnColorSpaceTransform.TCVN_CST_HLS_TO_RGB_FULL);
AddLocalEnumeration('TCVN_CST_LBGR_TO_LAB', ETcVnColorSpaceTransform.TCVN_CST_LBGR_TO_LAB);
AddLocalEnumeration('TCVN_CST_LRGB_TO_LAB', ETcVnColorSpaceTransform.TCVN_CST_LRGB_TO_LAB);
AddLocalEnumeration('TCVN_CST_LBGR_TO_LUV', ETcVnColorSpaceTransform.TCVN_CST_LBGR_TO_LUV);
AddLocalEnumeration('TCVN_CST_LRGB_TO_LUV', ETcVnColorSpaceTransform.TCVN_CST_LRGB_TO_LUV);
AddLocalEnumeration('TCVN_CST_LAB_TO_LBGR', ETcVnColorSpaceTransform.TCVN_CST_LAB_TO_LBGR);
AddLocalEnumeration('TCVN_CST_LAB_TO_LRGB', ETcVnColorSpaceTransform.TCVN_CST_LAB_TO_LRGB);
AddLocalEnumeration('TCVN_CST_LUV_TO_LBGR', ETcVnColorSpaceTransform.TCVN_CST_LUV_TO_LBGR);
AddLocalEnumeration('TCVN_CST_LUV_TO_LRGB', ETcVnColorSpaceTransform.TCVN_CST_LUV_TO_LRGB);
AddLocalEnumeration('TCVN_CST_BGR_TO_YUV', ETcVnColorSpaceTransform.TCVN_CST_BGR_TO_YUV);
AddLocalEnumeration('TCVN_CST_RGB_TO_YUV', ETcVnColorSpaceTransform.TCVN_CST_RGB_TO_YUV);
AddLocalEnumeration('TCVN_CST_YUV_TO_BGR', ETcVnColorSpaceTransform.TCVN_CST_YUV_TO_BGR);
AddLocalEnumeration('TCVN_CST_YUV_TO_RGB', ETcVnColorSpaceTransform.TCVN_CST_YUV_TO_RGB);
AddLocalEnumeration('TCVN_CST_BAYER_RG_TO_GRAY', ETcVnColorSpaceTransform.TCVN_CST_BAYER_RG_TO_GRAY);
AddLocalEnumeration('TCVN_CST_BAYER_GR_TO_GRAY', ETcVnColorSpaceTransform.TCVN_CST_BAYER_GR_TO_GRAY);
AddLocalEnumeration('TCVN_CST_BAYER_BG_TO_GRAY', ETcVnColorSpaceTransform.TCVN_CST_BAYER_BG_TO_GRAY);
AddLocalEnumeration('TCVN_CST_BAYER_GB_TO_GRAY', ETcVnColorSpaceTransform.TCVN_CST_BAYER_GB_TO_GRAY);
AddLocalEnumeration('TCVN_CST_YUV_420_NV12_TO_RGB', ETcVnColorSpaceTransform.TCVN_CST_YUV_420_NV12_TO_RGB);
AddLocalEnumeration('TCVN_CST_YUV_420_NV12_TO_BGR', ETcVnColorSpaceTransform.TCVN_CST_YUV_420_NV12_TO_BGR);
AddLocalEnumeration('TCVN_CST_YUV_420_NV21_TO_RGB', ETcVnColorSpaceTransform.TCVN_CST_YUV_420_NV21_TO_RGB);
AddLocalEnumeration('TCVN_CST_YUV_420_NV21_TO_BGR', ETcVnColorSpaceTransform.TCVN_CST_YUV_420_NV21_TO_BGR);
AddLocalEnumeration('TCVN_CST_YUV_420_SP_TO_RGB', ETcVnColorSpaceTransform.TCVN_CST_YUV_420_SP_TO_RGB);
AddLocalEnumeration('TCVN_CST_YUV_420_SP_TO_BGR', ETcVnColorSpaceTransform.TCVN_CST_YUV_420_SP_TO_BGR);
AddLocalEnumeration('TCVN_CST_YUV_420_NV12_TO_RGBA', ETcVnColorSpaceTransform.TCVN_CST_YUV_420_NV12_TO_RGBA);
AddLocalEnumeration('TCVN_CST_YUV_420_NV12_TO_BGRA', ETcVnColorSpaceTransform.TCVN_CST_YUV_420_NV12_TO_BGRA);
AddLocalEnumeration('TCVN_CST_YUV_420_NV21_TO_RGBA', ETcVnColorSpaceTransform.TCVN_CST_YUV_420_NV21_TO_RGBA);
AddLocalEnumeration('TCVN_CST_YUV_420_NV21_TO_BGRA', ETcVnColorSpaceTransform.TCVN_CST_YUV_420_NV21_TO_BGRA);
AddLocalEnumeration('TCVN_CST_YUV_420_SP_TO_RGBA', ETcVnColorSpaceTransform.TCVN_CST_YUV_420_SP_TO_RGBA);
AddLocalEnumeration('TCVN_CST_YUV_420_SP_TO_BGRA', ETcVnColorSpaceTransform.TCVN_CST_YUV_420_SP_TO_BGRA);
AddLocalEnumeration('TCVN_CST_YUV_420_YV12_TO_RGB', ETcVnColorSpaceTransform.TCVN_CST_YUV_420_YV12_TO_RGB);
AddLocalEnumeration('TCVN_CST_YUV_420_YV12_TO_BGR', ETcVnColorSpaceTransform.TCVN_CST_YUV_420_YV12_TO_BGR);
AddLocalEnumeration('TCVN_CST_YUV_420_IYUV_TO_RGB', ETcVnColorSpaceTransform.TCVN_CST_YUV_420_IYUV_TO_RGB);
AddLocalEnumeration('TCVN_CST_YUV_420_IYUV_TO_BGR', ETcVnColorSpaceTransform.TCVN_CST_YUV_420_IYUV_TO_BGR);
AddLocalEnumeration('TCVN_CST_YUV_420_I420_TO_RGB', ETcVnColorSpaceTransform.TCVN_CST_YUV_420_I420_TO_RGB);
AddLocalEnumeration('TCVN_CST_YUV_420_I420_TO_BGR', ETcVnColorSpaceTransform.TCVN_CST_YUV_420_I420_TO_BGR);
AddLocalEnumeration('TCVN_CST_YUV_420_P_TO_RGB', ETcVnColorSpaceTransform.TCVN_CST_YUV_420_P_TO_RGB);
AddLocalEnumeration('TCVN_CST_YUV_420_P_TO_BGR', ETcVnColorSpaceTransform.TCVN_CST_YUV_420_P_TO_BGR);
AddLocalEnumeration('TCVN_CST_YUV_420_YV12_TO_RGBA', ETcVnColorSpaceTransform.TCVN_CST_YUV_420_YV12_TO_RGBA);
AddLocalEnumeration('TCVN_CST_YUV_420_YV12_TO_BGRA', ETcVnColorSpaceTransform.TCVN_CST_YUV_420_YV12_TO_BGRA);
AddLocalEnumeration('TCVN_CST_YUV_420_IYUV_TO_RGBA', ETcVnColorSpaceTransform.TCVN_CST_YUV_420_IYUV_TO_RGBA);
AddLocalEnumeration('TCVN_CST_YUV_420_IYUV_TO_BGRA', ETcVnColorSpaceTransform.TCVN_CST_YUV_420_IYUV_TO_BGRA);
AddLocalEnumeration('TCVN_CST_YUV_420_I420_TO_RGBA', ETcVnColorSpaceTransform.TCVN_CST_YUV_420_I420_TO_RGBA);
AddLocalEnumeration('TCVN_CST_YUV_420_I420_TO_BGRA', ETcVnColorSpaceTransform.TCVN_CST_YUV_420_I420_TO_BGRA);
AddLocalEnumeration('TCVN_CST_YUV_420_P_TO_RGBA', ETcVnColorSpaceTransform.TCVN_CST_YUV_420_P_TO_RGBA);
AddLocalEnumeration('TCVN_CST_YUV_420_P_TO_BGRA', ETcVnColorSpaceTransform.TCVN_CST_YUV_420_P_TO_BGRA);
AddLocalEnumeration('TCVN_CST_YUV_420_TO_GRAY', ETcVnColorSpaceTransform.TCVN_CST_YUV_420_TO_GRAY);
AddLocalEnumeration('TCVN_CST_YUV_420_NV21_TO_GRAY', ETcVnColorSpaceTransform.TCVN_CST_YUV_420_NV21_TO_GRAY);
AddLocalEnumeration('TCVN_CST_YUV_420_NV12_TO_GRAY', ETcVnColorSpaceTransform.TCVN_CST_YUV_420_NV12_TO_GRAY);
AddLocalEnumeration('TCVN_CST_YUV_420_YV12_TO_GRAY', ETcVnColorSpaceTransform.TCVN_CST_YUV_420_YV12_TO_GRAY);
AddLocalEnumeration('TCVN_CST_YUV_420_IYUV_TO_GRAY', ETcVnColorSpaceTransform.TCVN_CST_YUV_420_IYUV_TO_GRAY);
AddLocalEnumeration('TCVN_CST_YUV_420_I420_TO_GRAY', ETcVnColorSpaceTransform.TCVN_CST_YUV_420_I420_TO_GRAY);
AddLocalEnumeration('TCVN_CST_YUV_420_SP_TO_GRAY', ETcVnColorSpaceTransform.TCVN_CST_YUV_420_SP_TO_GRAY);
AddLocalEnumeration('TCVN_CST_YUV_420_P_TO_GRAY', ETcVnColorSpaceTransform.TCVN_CST_YUV_420_P_TO_GRAY);
AddLocalEnumeration('TCVN_CST_YUV_422_UYVY_TO_RGB', ETcVnColorSpaceTransform.TCVN_CST_YUV_422_UYVY_TO_RGB);
AddLocalEnumeration('TCVN_CST_YUV_422_UYVY_TO_BGR', ETcVnColorSpaceTransform.TCVN_CST_YUV_422_UYVY_TO_BGR);
AddLocalEnumeration('TCVN_CST_YUV_422_Y422_TO_RGB', ETcVnColorSpaceTransform.TCVN_CST_YUV_422_Y422_TO_RGB);
AddLocalEnumeration('TCVN_CST_YUV_422_Y422_TO_BGR', ETcVnColorSpaceTransform.TCVN_CST_YUV_422_Y422_TO_BGR);
AddLocalEnumeration('TCVN_CST_YUV_422_UYNV_TO_RGB', ETcVnColorSpaceTransform.TCVN_CST_YUV_422_UYNV_TO_RGB);
AddLocalEnumeration('TCVN_CST_YUV_422_UYNV_TO_BGR', ETcVnColorSpaceTransform.TCVN_CST_YUV_422_UYNV_TO_BGR);
AddLocalEnumeration('TCVN_CST_YUV_422_UYVY_TO_RGBA', ETcVnColorSpaceTransform.TCVN_CST_YUV_422_UYVY_TO_RGBA);
AddLocalEnumeration('TCVN_CST_YUV_422_UYVY_TO_BGRA', ETcVnColorSpaceTransform.TCVN_CST_YUV_422_UYVY_TO_BGRA);
AddLocalEnumeration('TCVN_CST_YUV_422_Y422_TO_RGBA', ETcVnColorSpaceTransform.TCVN_CST_YUV_422_Y422_TO_RGBA);
AddLocalEnumeration('TCVN_CST_YUV_422_Y422_TO_BGRA', ETcVnColorSpaceTransform.TCVN_CST_YUV_422_Y422_TO_BGRA);
AddLocalEnumeration('TCVN_CST_YUV_422_UYNV_TO_RGBA', ETcVnColorSpaceTransform.TCVN_CST_YUV_422_UYNV_TO_RGBA);
AddLocalEnumeration('TCVN_CST_YUV_422_UYNV_TO_BGRA', ETcVnColorSpaceTransform.TCVN_CST_YUV_422_UYNV_TO_BGRA);
AddLocalEnumeration('TCVN_CST_YUV_422_YUY2_TO_RGB', ETcVnColorSpaceTransform.TCVN_CST_YUV_422_YUY2_TO_RGB);
AddLocalEnumeration('TCVN_CST_YUV_422_YUY2_TO_BGR', ETcVnColorSpaceTransform.TCVN_CST_YUV_422_YUY2_TO_BGR);
AddLocalEnumeration('TCVN_CST_YUV_422_YVYU_TO_RGB', ETcVnColorSpaceTransform.TCVN_CST_YUV_422_YVYU_TO_RGB);
AddLocalEnumeration('TCVN_CST_YUV_422_YVYU_TO_BGR', ETcVnColorSpaceTransform.TCVN_CST_YUV_422_YVYU_TO_BGR);
AddLocalEnumeration('TCVN_CST_YUV_422_YUYV_TO_RGB', ETcVnColorSpaceTransform.TCVN_CST_YUV_422_YUYV_TO_RGB);
AddLocalEnumeration('TCVN_CST_YUV_422_YUYV_TO_BGR', ETcVnColorSpaceTransform.TCVN_CST_YUV_422_YUYV_TO_BGR);
AddLocalEnumeration('TCVN_CST_YUV_422_YUNV_TO_RGB', ETcVnColorSpaceTransform.TCVN_CST_YUV_422_YUNV_TO_RGB);
AddLocalEnumeration('TCVN_CST_YUV_422_YUNV_TO_BGR', ETcVnColorSpaceTransform.TCVN_CST_YUV_422_YUNV_TO_BGR);
AddLocalEnumeration('TCVN_CST_YUV_422_YUY2_TO_RGBA', ETcVnColorSpaceTransform.TCVN_CST_YUV_422_YUY2_TO_RGBA);
AddLocalEnumeration('TCVN_CST_YUV_422_YUY2_TO_BGRA', ETcVnColorSpaceTransform.TCVN_CST_YUV_422_YUY2_TO_BGRA);
AddLocalEnumeration('TCVN_CST_YUV_422_YVYU_TO_RGBA', ETcVnColorSpaceTransform.TCVN_CST_YUV_422_YVYU_TO_RGBA);
AddLocalEnumeration('TCVN_CST_YUV_422_YVYU_TO_BGRA', ETcVnColorSpaceTransform.TCVN_CST_YUV_422_YVYU_TO_BGRA);
AddLocalEnumeration('TCVN_CST_YUV_422_YUYV_TO_RGBA', ETcVnColorSpaceTransform.TCVN_CST_YUV_422_YUYV_TO_RGBA);
AddLocalEnumeration('TCVN_CST_YUV_422_YUYV_TO_BGRA', ETcVnColorSpaceTransform.TCVN_CST_YUV_422_YUYV_TO_BGRA);
AddLocalEnumeration('TCVN_CST_YUV_422_YUNV_TO_RGBA', ETcVnColorSpaceTransform.TCVN_CST_YUV_422_YUNV_TO_RGBA);
AddLocalEnumeration('TCVN_CST_YUV_422_YUNV_TO_BGRA', ETcVnColorSpaceTransform.TCVN_CST_YUV_422_YUNV_TO_BGRA);
AddLocalEnumeration('TCVN_CST_YUV_422_UYVY_TO_GRAY', ETcVnColorSpaceTransform.TCVN_CST_YUV_422_UYVY_TO_GRAY);
AddLocalEnumeration('TCVN_CST_YUV_422_YUY2_TO_GRAY', ETcVnColorSpaceTransform.TCVN_CST_YUV_422_YUY2_TO_GRAY);
AddLocalEnumeration('TCVN_CST_YUV_422_Y422_TO_GRAY', ETcVnColorSpaceTransform.TCVN_CST_YUV_422_Y422_TO_GRAY);
AddLocalEnumeration('TCVN_CST_YUV_422_UYNV_TO_GRAY', ETcVnColorSpaceTransform.TCVN_CST_YUV_422_UYNV_TO_GRAY);
AddLocalEnumeration('TCVN_CST_YUV_422_YVYU_TO_GRAY', ETcVnColorSpaceTransform.TCVN_CST_YUV_422_YVYU_TO_GRAY);
AddLocalEnumeration('TCVN_CST_YUV_422_YUYV_TO_GRAY', ETcVnColorSpaceTransform.TCVN_CST_YUV_422_YUYV_TO_GRAY);
AddLocalEnumeration('TCVN_CST_YUV_422_YUNV_TO_GRAY', ETcVnColorSpaceTransform.TCVN_CST_YUV_422_YUNV_TO_GRAY);
AddLocalEnumeration('TCVN_CST_RGBA_TO_PREMULTIPLICATED_RGBA', ETcVnColorSpaceTransform.TCVN_CST_RGBA_TO_PREMULTIPLICATED_RGBA);
AddLocalEnumeration('TCVN_CST_PREMULTIPLICATED_RGBA_TO_RGBA', ETcVnColorSpaceTransform.TCVN_CST_PREMULTIPLICATED_RGBA_TO_RGBA);
AddLocalEnumeration('TCVN_CST_RGB_TO_YUV_420_I420', ETcVnColorSpaceTransform.TCVN_CST_RGB_TO_YUV_420_I420);
AddLocalEnumeration('TCVN_CST_BGR_TO_YUV_420_I420', ETcVnColorSpaceTransform.TCVN_CST_BGR_TO_YUV_420_I420);
AddLocalEnumeration('TCVN_CST_RGB_TO_YUV_420_IYUV', ETcVnColorSpaceTransform.TCVN_CST_RGB_TO_YUV_420_IYUV);
AddLocalEnumeration('TCVN_CST_BGR_TO_YUV_420_IYUV', ETcVnColorSpaceTransform.TCVN_CST_BGR_TO_YUV_420_IYUV);
AddLocalEnumeration('TCVN_CST_RGBA_TO_YUV_420_I420', ETcVnColorSpaceTransform.TCVN_CST_RGBA_TO_YUV_420_I420);
AddLocalEnumeration('TCVN_CST_BGRA_TO_YUV_420_I420', ETcVnColorSpaceTransform.TCVN_CST_BGRA_TO_YUV_420_I420);
AddLocalEnumeration('TCVN_CST_RGBA_TO_YUV_420_IYUV', ETcVnColorSpaceTransform.TCVN_CST_RGBA_TO_YUV_420_IYUV);
AddLocalEnumeration('TCVN_CST_BGRA_TO_YUV_420_IYUV', ETcVnColorSpaceTransform.TCVN_CST_BGRA_TO_YUV_420_IYUV);
AddLocalEnumeration('TCVN_CST_RGB_TO_YUV_420_YV12', ETcVnColorSpaceTransform.TCVN_CST_RGB_TO_YUV_420_YV12);
AddLocalEnumeration('TCVN_CST_BGR_TO_YUV_420_YV12', ETcVnColorSpaceTransform.TCVN_CST_BGR_TO_YUV_420_YV12);
AddLocalEnumeration('TCVN_CST_RGBA_TO_YUV_420_YV12', ETcVnColorSpaceTransform.TCVN_CST_RGBA_TO_YUV_420_YV12);
AddLocalEnumeration('TCVN_CST_BGRA_TO_YUV_420_YV12', ETcVnColorSpaceTransform.TCVN_CST_BGRA_TO_YUV_420_YV12);
AddLocalEnumeration('TCVN_CST_BAYER_RG_TO_BGR_EA', ETcVnColorSpaceTransform.TCVN_CST_BAYER_RG_TO_BGR_EA);
AddLocalEnumeration('TCVN_CST_BAYER_GR_TO_BGR_EA', ETcVnColorSpaceTransform.TCVN_CST_BAYER_GR_TO_BGR_EA);
AddLocalEnumeration('TCVN_CST_BAYER_BG_TO_BGR_EA', ETcVnColorSpaceTransform.TCVN_CST_BAYER_BG_TO_BGR_EA);
AddLocalEnumeration('TCVN_CST_BAYER_GB_TO_BGR_EA', ETcVnColorSpaceTransform.TCVN_CST_BAYER_GB_TO_BGR_EA);
AddLocalEnumeration('TCVN_CST_BAYER_RG_TO_RGB_EA', ETcVnColorSpaceTransform.TCVN_CST_BAYER_RG_TO_RGB_EA);
AddLocalEnumeration('TCVN_CST_BAYER_GR_TO_RGB_EA', ETcVnColorSpaceTransform.TCVN_CST_BAYER_GR_TO_RGB_EA);
AddLocalEnumeration('TCVN_CST_BAYER_BG_TO_RGB_EA', ETcVnColorSpaceTransform.TCVN_CST_BAYER_BG_TO_RGB_EA);
AddLocalEnumeration('TCVN_CST_BAYER_GB_TO_RGB_EA', ETcVnColorSpaceTransform.TCVN_CST_BAYER_GB_TO_RGB_EA);
AddLocalEnumeration('TCVN_CST_BAYER_RG_TO_BGRA', ETcVnColorSpaceTransform.TCVN_CST_BAYER_RG_TO_BGRA);
AddLocalEnumeration('TCVN_CST_BAYER_GR_TO_BGRA', ETcVnColorSpaceTransform.TCVN_CST_BAYER_GR_TO_BGRA);
AddLocalEnumeration('TCVN_CST_BAYER_BG_TO_BGRA', ETcVnColorSpaceTransform.TCVN_CST_BAYER_BG_TO_BGRA);
AddLocalEnumeration('TCVN_CST_BAYER_GB_TO_BGRA', ETcVnColorSpaceTransform.TCVN_CST_BAYER_GB_TO_BGRA);
AddLocalEnumeration('TCVN_CST_BAYER_RG_TO_RGBA', ETcVnColorSpaceTransform.TCVN_CST_BAYER_RG_TO_RGBA);
AddLocalEnumeration('TCVN_CST_BAYER_GR_TO_RGBA', ETcVnColorSpaceTransform.TCVN_CST_BAYER_GR_TO_RGBA);
AddLocalEnumeration('TCVN_CST_BAYER_BG_TO_RGBA', ETcVnColorSpaceTransform.TCVN_CST_BAYER_BG_TO_RGBA);
AddLocalEnumeration('TCVN_CST_BAYER_GB_TO_RGBA', ETcVnColorSpaceTransform.TCVN_CST_BAYER_GB_TO_RGBA);
AddLocalEnumeration('TCVN_CST_MAX', ETcVnColorSpaceTransform.TCVN_CST_MAX);
END_METHOD

PROPERTY PUBLIC Identifier : T_MAXSTRING
GET
Identifier := 'ETcVnColorSpaceTransform';
END_GET
END_PROPERTY

METHOD IsEnumeratorValueEqual : BOOL
VAR_INPUT
	Enumerator : I_KeyValueForwardEnumerator;
END_VAR
VAR
	storedValue : ETcVnColorSpaceTransform;
END_VAR
IF NOT Enumerator.TryGet(storedValue) THEN
	RETURN;
END_IF

IsEnumeratorValueEqual := storedValue = activeData;
END_METHOD

METHOD PUBLIC MakeReferenceTo
VAR_INPUT
	ReferenceTarget : REFERENCE TO ETcVnColorSpaceTransform;
END_VAR
activeData REF= ReferenceTarget;
SetBaseDatatypeReference();
END_METHOD

METHOD PROTECTED SetBaseDatatypeReference
VAR_INPUT
END_VAR
enumBaseDatatype.MakeReferenceTo(activeData);
END_METHOD

PROPERTY PUBLIC Size : UDINT
GET
Size := SIZEOF(activeData);
END_GET
END_PROPERTY

METHOD TryMakeReferenceTo : BOOL
VAR_INPUT
	Target : I_Datatype;
END_VAR
VAR
	targetAsEnum : I_EnumDatatype;
	pTargetData : POINTER TO ETcVnColorSpaceTransform;
END_VAR
IF NOT Target.TryResolveAsEnumDatatype(targetAsEnum) THEN
	RETURN;
END_IF

IF targetAsEnum.Identifier <> Identifier THEN
	RETURN;
END_IF

pTargetData := Target.Address;
activeData REF= pTargetData^;
SetBaseDatatypeReference();
TryMakeReferenceTo := TRUE;
END_METHOD

PROPERTY PUBLIC Value : ETcVnColorSpaceTransform
GET
Value := activeData;
END_GET
SET
activeData := Value;
END_SET
END_PROPERTY

END_FUNCTION_BLOCK

// ---- Enums/_ETcVnPixelPackMode.TcPOU
{attribute 'linkalways'} 
{attribute 'no_explicit_call' := 'This FB is a CLASS and must be accessed using methods or properties'}
{attribute 'enable_dynamic_creation'}
FUNCTION_BLOCK _ETcVnPixelPackMode EXTENDS EnumDatatypeBase
VAR
	localData : ETcVnPixelPackMode;
	activeData : REFERENCE TO ETcVnPixelPackMode;
	enumBaseDatatype : _BYTE(localData);
END_VAR

METHOD PRIVATE AddLocalEnumeration
VAR_INPUT
	Enumeration : T_MAXSTRING;
	Value : ETcVnPixelPackMode;
END_VAR
AddEnumeration(Enumeration, Value);
END_METHOD

PROPERTY PUBLIC Address : PVOID
GET
Address := ADR(activeData);
END_GET
END_PROPERTY

METHOD PUBLIC ClearReference
VAR_INPUT
END_VAR
activeData REF= localData;
SetBaseDatatypeReference();
END_METHOD

METHOD PUBLIC Clone : I_Datatype
VAR
    pClone : POINTER TO _ETcVnPixelPackMode;
END_VAR
pClone := __NEW(_ETcVnPixelPackMode(InitialValue := Value));
Clone := pClone^;
END_METHOD

METHOD FB_init : BOOL
VAR_INPUT
	bInitRetains : BOOL; // if TRUE, the retain variables are initialized (warm start / cold start)
	bInCopyCode : BOOL;  // if TRUE, the instance afterwards gets moved into the copy code (online change)
	InitialValue : ETcVnPixelPackMode;
END_VAR
localData := InitialValue;
AddBaseDatatype(enumBaseDatatype);
ClearReference();

AddLocalEnumeration('TCVN_PPM_NONE', ETcVnPixelPackMode.TCVN_PPM_NONE);
AddLocalEnumeration('TCVN_PPM_MONO1P', ETcVnPixelPackMode.TCVN_PPM_MONO1P);
AddLocalEnumeration('TCVN_PPM_MONO2P', ETcVnPixelPackMode.TCVN_PPM_MONO2P);
AddLocalEnumeration('TCVN_PPM_MONO4P', ETcVnPixelPackMode.TCVN_PPM_MONO4P);
AddLocalEnumeration('TCVN_PPM_MONO10PACKED', ETcVnPixelPackMode.TCVN_PPM_MONO10PACKED);
AddLocalEnumeration('TCVN_PPM_MONO12PACKED', ETcVnPixelPackMode.TCVN_PPM_MONO12PACKED);
AddLocalEnumeration('TCVN_PPM_RGB10V1PACKED', ETcVnPixelPackMode.TCVN_PPM_RGB10V1PACKED);
AddLocalEnumeration('TCVN_PPM_RGB10P32', ETcVnPixelPackMode.TCVN_PPM_RGB10P32);
AddLocalEnumeration('TCVN_PPM_RGB12V1PACKED', ETcVnPixelPackMode.TCVN_PPM_RGB12V1PACKED);
AddLocalEnumeration('TCVN_PPM_RGB565P', ETcVnPixelPackMode.TCVN_PPM_RGB565P);
AddLocalEnumeration('TCVN_PPM_BGR565P', ETcVnPixelPackMode.TCVN_PPM_BGR565P);
AddLocalEnumeration('TCVN_PPM_MONO10P', ETcVnPixelPackMode.TCVN_PPM_MONO10P);
AddLocalEnumeration('TCVN_PPM_MONO12P', ETcVnPixelPackMode.TCVN_PPM_MONO12P);
END_METHOD

PROPERTY PUBLIC Identifier : T_MAXSTRING
GET
Identifier := 'ETcVnPixelPackMode';
END_GET
END_PROPERTY

METHOD IsEnumeratorValueEqual : BOOL
VAR_INPUT
	Enumerator : I_KeyValueForwardEnumerator;
END_VAR
VAR
	storedValue : ETcVnPixelPackMode;
END_VAR
IF NOT Enumerator.TryGet(storedValue) THEN
	RETURN;
END_IF

IsEnumeratorValueEqual := storedValue = activeData;
END_METHOD

METHOD PUBLIC MakeReferenceTo
VAR_INPUT
	ReferenceTarget : REFERENCE TO ETcVnPixelPackMode;
END_VAR
activeData REF= ReferenceTarget;
SetBaseDatatypeReference();
END_METHOD

METHOD PROTECTED SetBaseDatatypeReference
VAR_INPUT
END_VAR
enumBaseDatatype.MakeReferenceTo(activeData);
END_METHOD

PROPERTY PUBLIC Size : UDINT
GET
Size := SIZEOF(activeData);
END_GET
END_PROPERTY

METHOD TryMakeReferenceTo : BOOL
VAR_INPUT
	Target : I_Datatype;
END_VAR
VAR
	targetAsEnum : I_EnumDatatype;
	pTargetData : POINTER TO ETcVnPixelPackMode;
END_VAR
IF NOT Target.TryResolveAsEnumDatatype(targetAsEnum) THEN
	RETURN;
END_IF

IF targetAsEnum.Identifier <> Identifier THEN
	RETURN;
END_IF

pTargetData := Target.Address;
activeData REF= pTargetData^;
SetBaseDatatypeReference();
TryMakeReferenceTo := TRUE;
END_METHOD

PROPERTY PUBLIC Value : ETcVnPixelPackMode
GET
Value := activeData;
END_GET
SET
activeData := Value;
END_SET
END_PROPERTY

END_FUNCTION_BLOCK

// ---- Enums/_ETcVnPrototypeClusterer.TcPOU
{attribute 'linkalways'} 
{attribute 'no_explicit_call' := 'This FB is a CLASS and must be accessed using methods or properties'}
{attribute 'enable_dynamic_creation'}
FUNCTION_BLOCK _ETcVnPrototypeClusterer EXTENDS EnumDatatypeBase
VAR
	localData : ETcVnPrototypeClusterer;
	activeData : REFERENCE TO ETcVnPrototypeClusterer;
	enumBaseDatatype : _UDINT(localData);
END_VAR

METHOD PRIVATE AddLocalEnumeration
VAR_INPUT
	Enumeration : T_MAXSTRING;
	Value : ETcVnPrototypeClusterer;
END_VAR
AddEnumeration(Enumeration, Value);
END_METHOD

PROPERTY PUBLIC Address : PVOID
GET
Address := ADR(activeData);
END_GET
END_PROPERTY

METHOD PUBLIC ClearReference
VAR_INPUT
END_VAR
activeData REF= localData;
SetBaseDatatypeReference();
END_METHOD

METHOD PUBLIC Clone : I_Datatype
VAR
    pClone : POINTER TO _ETcVnPrototypeClusterer;
END_VAR
pClone := __NEW(_ETcVnPrototypeClusterer(InitialValue := Value));
Clone := pClone^;
END_METHOD

METHOD FB_init : BOOL
VAR_INPUT
	bInitRetains : BOOL; // if TRUE, the retain variables are initialized (warm start / cold start)
	bInCopyCode : BOOL;  // if TRUE, the instance afterwards gets moved into the copy code (online change)
	InitialValue : ETcVnPrototypeClusterer;
END_VAR
localData := InitialValue;
AddBaseDatatype(enumBaseDatatype);
ClearReference();

AddLocalEnumeration('TCVN_PC_NOVELTY_DETECTOR', ETcVnPrototypeClusterer.TCVN_PC_NOVELTY_DETECTOR);
AddLocalEnumeration('TCVN_PC_CLUSTERER', ETcVnPrototypeClusterer.TCVN_PC_CLUSTERER);
END_METHOD

PROPERTY PUBLIC Identifier : T_MAXSTRING
GET
Identifier := 'ETcVnPrototypeClusterer';
END_GET
END_PROPERTY

METHOD IsEnumeratorValueEqual : BOOL
VAR_INPUT
	Enumerator : I_KeyValueForwardEnumerator;
END_VAR
VAR
	storedValue : ETcVnPrototypeClusterer;
END_VAR
IF NOT Enumerator.TryGet(storedValue) THEN
	RETURN;
END_IF

IsEnumeratorValueEqual := storedValue = activeData;
END_METHOD

METHOD PUBLIC MakeReferenceTo
VAR_INPUT
	ReferenceTarget : REFERENCE TO ETcVnPrototypeClusterer;
END_VAR
activeData REF= ReferenceTarget;
SetBaseDatatypeReference();
END_METHOD

METHOD PROTECTED SetBaseDatatypeReference
VAR_INPUT
END_VAR
enumBaseDatatype.MakeReferenceTo(activeData);
END_METHOD

PROPERTY PUBLIC Size : UDINT
GET
Size := SIZEOF(activeData);
END_GET
END_PROPERTY

METHOD TryMakeReferenceTo : BOOL
VAR_INPUT
	Target : I_Datatype;
END_VAR
VAR
	targetAsEnum : I_EnumDatatype;
	pTargetData : POINTER TO ETcVnPrototypeClusterer;
END_VAR
IF NOT Target.TryResolveAsEnumDatatype(targetAsEnum) THEN
	RETURN;
END_IF

IF targetAsEnum.Identifier <> Identifier THEN
	RETURN;
END_IF

pTargetData := Target.Address;
activeData REF= pTargetData^;
SetBaseDatatypeReference();
TryMakeReferenceTo := TRUE;
END_METHOD

PROPERTY PUBLIC Value : ETcVnPrototypeClusterer
GET
Value := activeData;
END_GET
SET
activeData := Value;
END_SET
END_PROPERTY

END_FUNCTION_BLOCK

// ---- Enums/_ETcVnRectangleIntersection.TcPOU
{attribute 'linkalways'} 
{attribute 'no_explicit_call' := 'This FB is a CLASS and must be accessed using methods or properties'}
{attribute 'enable_dynamic_creation'}
FUNCTION_BLOCK _ETcVnRectangleIntersection EXTENDS EnumDatatypeBase
VAR
	localData : ETcVnRectangleIntersection;
	activeData : REFERENCE TO ETcVnRectangleIntersection;
	enumBaseDatatype : _DINT(localData);
END_VAR

METHOD PRIVATE AddLocalEnumeration
VAR_INPUT
	Enumeration : T_MAXSTRING;
	Value : ETcVnRectangleIntersection;
END_VAR
AddEnumeration(Enumeration, Value);
END_METHOD

PROPERTY PUBLIC Address : PVOID
GET
Address := ADR(activeData);
END_GET
END_PROPERTY

METHOD PUBLIC ClearReference
VAR_INPUT
END_VAR
activeData REF= localData;
SetBaseDatatypeReference();
END_METHOD

METHOD PUBLIC Clone : I_Datatype
VAR
    pClone : POINTER TO _ETcVnRectangleIntersection;
END_VAR
pClone := __NEW(_ETcVnRectangleIntersection(InitialValue := Value));
Clone := pClone^;
END_METHOD

METHOD FB_init : BOOL
VAR_INPUT
	bInitRetains : BOOL; // if TRUE, the retain variables are initialized (warm start / cold start)
	bInCopyCode : BOOL;  // if TRUE, the instance afterwards gets moved into the copy code (online change)
	InitialValue : ETcVnRectangleIntersection;
END_VAR
localData := InitialValue;
AddBaseDatatype(enumBaseDatatype);
ClearReference();

AddLocalEnumeration('TCVN_RI_NONE', ETcVnRectangleIntersection.TCVN_RI_NONE);
AddLocalEnumeration('TCVN_RI_PARTIAL', ETcVnRectangleIntersection.TCVN_RI_PARTIAL);
AddLocalEnumeration('TCVN_RI_FULL', ETcVnRectangleIntersection.TCVN_RI_FULL);
END_METHOD

PROPERTY PUBLIC Identifier : T_MAXSTRING
GET
Identifier := 'ETcVnRectangleIntersection';
END_GET
END_PROPERTY

METHOD IsEnumeratorValueEqual : BOOL
VAR_INPUT
	Enumerator : I_KeyValueForwardEnumerator;
END_VAR
VAR
	storedValue : ETcVnRectangleIntersection;
END_VAR
IF NOT Enumerator.TryGet(storedValue) THEN
	RETURN;
END_IF

IsEnumeratorValueEqual := storedValue = activeData;
END_METHOD

METHOD PUBLIC MakeReferenceTo
VAR_INPUT
	ReferenceTarget : REFERENCE TO ETcVnRectangleIntersection;
END_VAR
activeData REF= ReferenceTarget;
SetBaseDatatypeReference();
END_METHOD

METHOD PROTECTED SetBaseDatatypeReference
VAR_INPUT
END_VAR
enumBaseDatatype.MakeReferenceTo(activeData);
END_METHOD

PROPERTY PUBLIC Size : UDINT
GET
Size := SIZEOF(activeData);
END_GET
END_PROPERTY

METHOD TryMakeReferenceTo : BOOL
VAR_INPUT
	Target : I_Datatype;
END_VAR
VAR
	targetAsEnum : I_EnumDatatype;
	pTargetData : POINTER TO ETcVnRectangleIntersection;
END_VAR
IF NOT Target.TryResolveAsEnumDatatype(targetAsEnum) THEN
	RETURN;
END_IF

IF targetAsEnum.Identifier <> Identifier THEN
	RETURN;
END_IF

pTargetData := Target.Address;
activeData REF= pTargetData^;
SetBaseDatatypeReference();
TryMakeReferenceTo := TRUE;
END_METHOD

PROPERTY PUBLIC Value : ETcVnRectangleIntersection
GET
Value := activeData;
END_GET
SET
activeData := Value;
END_SET
END_PROPERTY

END_FUNCTION_BLOCK

// ---- Enums/_ETcVnRotationAngle.TcPOU
{attribute 'linkalways'} 
{attribute 'no_explicit_call' := 'This FB is a CLASS and must be accessed using methods or properties'}
{attribute 'enable_dynamic_creation'}
FUNCTION_BLOCK _ETcVnRotationAngle EXTENDS EnumDatatypeBase
VAR
	localData : ETcVnRotationAngle;
	activeData : REFERENCE TO ETcVnRotationAngle;
	enumBaseDatatype : _DINT(localData);
END_VAR

METHOD PRIVATE AddLocalEnumeration
VAR_INPUT
	Enumeration : T_MAXSTRING;
	Value : ETcVnRotationAngle;
END_VAR
AddEnumeration(Enumeration, Value);
END_METHOD

PROPERTY PUBLIC Address : PVOID
GET
Address := ADR(activeData);
END_GET
END_PROPERTY

METHOD PUBLIC ClearReference
VAR_INPUT
END_VAR
activeData REF= localData;
SetBaseDatatypeReference();
END_METHOD

METHOD PUBLIC Clone : I_Datatype
VAR
    pClone : POINTER TO _ETcVnRotationAngle;
END_VAR
pClone := __NEW(_ETcVnRotationAngle(InitialValue := Value));
Clone := pClone^;
END_METHOD

METHOD FB_init : BOOL
VAR_INPUT
	bInitRetains : BOOL; // if TRUE, the retain variables are initialized (warm start / cold start)
	bInCopyCode : BOOL;  // if TRUE, the instance afterwards gets moved into the copy code (online change)
	InitialValue : ETcVnRotationAngle;
END_VAR
localData := InitialValue;
AddBaseDatatype(enumBaseDatatype);
ClearReference();

AddLocalEnumeration('TCVN_RA_90_DEG', ETcVnRotationAngle.TCVN_RA_90_DEG);
AddLocalEnumeration('TCVN_RA_180_DEG', ETcVnRotationAngle.TCVN_RA_180_DEG);
AddLocalEnumeration('TCVN_RA_270_DEG', ETcVnRotationAngle.TCVN_RA_270_DEG);
END_METHOD

PROPERTY PUBLIC Identifier : T_MAXSTRING
GET
Identifier := 'ETcVnRotationAngle';
END_GET
END_PROPERTY

METHOD IsEnumeratorValueEqual : BOOL
VAR_INPUT
	Enumerator : I_KeyValueForwardEnumerator;
END_VAR
VAR
	storedValue : ETcVnRotationAngle;
END_VAR
IF NOT Enumerator.TryGet(storedValue) THEN
	RETURN;
END_IF

IsEnumeratorValueEqual := storedValue = activeData;
END_METHOD

METHOD PUBLIC MakeReferenceTo
VAR_INPUT
	ReferenceTarget : REFERENCE TO ETcVnRotationAngle;
END_VAR
activeData REF= ReferenceTarget;
SetBaseDatatypeReference();
END_METHOD

METHOD PROTECTED SetBaseDatatypeReference
VAR_INPUT
END_VAR
enumBaseDatatype.MakeReferenceTo(activeData);
END_METHOD

PROPERTY PUBLIC Size : UDINT
GET
Size := SIZEOF(activeData);
END_GET
END_PROPERTY

METHOD TryMakeReferenceTo : BOOL
VAR_INPUT
	Target : I_Datatype;
END_VAR
VAR
	targetAsEnum : I_EnumDatatype;
	pTargetData : POINTER TO ETcVnRotationAngle;
END_VAR
IF NOT Target.TryResolveAsEnumDatatype(targetAsEnum) THEN
	RETURN;
END_IF

IF targetAsEnum.Identifier <> Identifier THEN
	RETURN;
END_IF

pTargetData := Target.Address;
activeData REF= pTargetData^;
SetBaseDatatypeReference();
TryMakeReferenceTo := TRUE;
END_METHOD

PROPERTY PUBLIC Value : ETcVnRotationAngle
GET
Value := activeData;
END_GET
SET
activeData := Value;
END_SET
END_PROPERTY

END_FUNCTION_BLOCK

// ---- Enums/_ETcVnRTrees.TcPOU
{attribute 'linkalways'} 
{attribute 'no_explicit_call' := 'This FB is a CLASS and must be accessed using methods or properties'}
{attribute 'enable_dynamic_creation'}
FUNCTION_BLOCK _ETcVnRTrees EXTENDS EnumDatatypeBase
VAR
	localData : ETcVnRTrees;
	activeData : REFERENCE TO ETcVnRTrees;
	enumBaseDatatype : _UDINT(localData);
END_VAR

METHOD PRIVATE AddLocalEnumeration
VAR_INPUT
	Enumeration : T_MAXSTRING;
	Value : ETcVnRTrees;
END_VAR
AddEnumeration(Enumeration, Value);
END_METHOD

PROPERTY PUBLIC Address : PVOID
GET
Address := ADR(activeData);
END_GET
END_PROPERTY

